// TwinCAT 3 PLC project _243401_DIOSNA_PLC
// ProgramVersion: 3.1.4026.19
// libraries:
//   Tc2_ControllerToolbox, * (Beckhoff Automation GmbH)
//   Tc2_Standard, * (Beckhoff Automation GmbH)
//   Tc2_SUPS, * (Beckhoff Automation GmbH)
//   Tc2_System, * (Beckhoff Automation GmbH)
//   Tc2_Utilities, * (Beckhoff Automation GmbH)
//   Tc3_Database, * (Beckhoff Automation GmbH)
//   Tc3_EventLogger, * (Beckhoff Automation GmbH)
//   Tc3_IPCDiag, * (Beckhoff Automation GmbH)
//   Tc3_Module, * (Beckhoff Automation GmbH)
// project tree:
//   DUTs/DataBase/ ST_BatchTrail.TcDUT, ST_ProcessData.TcDUT, ST_ShortData.TcDUT, ST_SPData.TcDUT
//   DUTs/Devices/ ST_Interface_CoilCtrl.TcDUT, ST_Interface_MotorCoilsCtrl.TcDUT, ST_Interface_MotorCtrl.TcDUT, ST_Interface_ValveCtrl.TcDUT
//   DUTs/ EN_Events.TcDUT, EN_RecipeType.TcDUT (not stored), ST_Alarm.TcDUT, ST_Batch.TcDUT, ST_Diagnostic.TcDUT, ST_HMI.TcDUT, ST_Control.TcDUT, ST_HMI_Time.TcDUT (not stored), ST_Interface_PidCtrl.TcDUT, ST_ProcessCmd2.TcDUT, ST_ProcessCmd.TcDUT, ST_PythonHandshake.TcDUT, ST_RecipeList.TcDUT (not stored), ST_RecipeSP.TcDUT, ST_Report.TcDUT, ST_RX_Python.TcDUT, ST_SeqControl.TcDUT, ST_Settings.TcDUT, ST_SP_ProcessCmd.TcDUT, ST_Time.TcDUT (not stored), ST_ToHMI.TcDUT, ST_Trend.TcDUT, ST_TX_Python.TcDUT
//   DUTs/Recipe/ ST_Cleaning_Phases.TcDUT, ST_Production_Phases.TcDUT, ST_RecipeInfo.TcDUT, ST_Recipe_Cleaning.TcDUT, ST_Recipe_Production.TcDUT
//   DUTs/ST_HMI/ ST_AlarmControl.TcDUT (not stored), ST_BatchControl.TcDUT, ST_MachineControl.TcDUT, ST_ProcessControl.TcDUT, ST_ReportControl.TcDUT
//   DUTs/ST_Mapping/ ST_EL1819.TcDUT, ST_EL2809.TcDUT, ST_EL3174.TcDUT, ST_EL4008.TcDUT, ST_EL4124.TcDUT, ST_EL9110.TcDUT
//   DUTs/ST_toHMI/ ST_EnableControl.TcDUT, ST_Header.TcDUT, ST_PID.TcDUT, ST_Prompts.TcDUT, ST_SP.TcDUT
//   FBs/Devices/ FB_AnalogInput.TcPOU, FB_AnalogOutput_v01.TcPOU, FB_AnalogOutput_v02.TcPOU, FB_CoilCtrl.TcPOU, FB_MotorCoilsCtrl.TcPOU, FB_MotorFreqCtrl.TcPOU, FB_PID.TcPOU, FB_PID_AutoTuner.TcPOU, FB_PID_Gain2Time.TcPOU, FB_PID_PWM.TcPOU, FB_TemperatureInput.TcPOU, FB_ValveCtrl32.TcPOU, FB_ValveCtrl52.TcPOU
//   FBs/ FB_AlarmDiagnostic.TcPOU, FB_AuditTrail_Write.TcPOU, FB_AVG200.TcPOU, FB_Batch.TcPOU, FB_BatchLog.TcPOU, FB_DeleteOldestFile.TcPOU, FB_FileSaveAs.TcPOU (not stored), FB_FileSaveAs_V02.TcPOU (not stored), FB_PythonScript.TcPOU, FB_Scale.TcPOU (not stored), FB_SystemDateTime.TcPOU, FB_TimeElapsed_HMI.TcPOU (not stored), FB_TONP.TcPOU (not stored)
//   Functions/ F_Interlocks.TcPOU (not stored), F_OperationalTime.TcPOU (not stored), F_Select.TcPOU, F_StepCMP.TcPOU (not stored), F_TimeBarHMI.TcPOU (not stored), F_TimerEt2String.TcPOU, F_TimerHMI.TcPOU (not stored), F_ToArrAlarms.TcPOU, F_ToArrInterlocks.TcPOU
//   GVLs/ CONST.TcGVL, GV.TcGVL, IN.TcGVL, OUT.TcGVL, Recipes.TcGVL
//   / PlcTask.TcTTO
//   POUs/0. Input/ P0_01_Mapping.TcPOU, P0_00_MAIN.TcPOU, P0_02_AnalogInput.TcPOU
//   POUs/1. Main Control/ P1_00_MAIN.TcPOU, P1_01_Recipe.TcPOU, P1_02_Batch.TcPOU, P1_03_Alarms.TcPOU, P1_04_MachineControl.TcPOU
//   POUs/2. Process/Cleaning/ _BlowingOut.TcPOU, _Control.TcPOU, _Draining.TcPOU, _MainCleaning.TcPOU, _PreCleaning.TcPOU, _PWCleaning.TcPOU, _Rinsing.TcPOU
//   POUs/2. Process/ P2_00_MAIN.TcPOU, P2_01_Production_Seq.TcPOU, P2_02_Cleaning_Seq.TcPOU, P2_03_Production_Ctrl.TcPOU, P2_04_Cleaning_Ctrl.TcPOU, P2_05_Process_Ctrl.TcPOU, P2_05_SP_Process_Ctrl.TcPOU, P2_06_Device_Ctrl.TcPOU, _Chopper.TcPOU, _FilterClean.TcPOU, _Mixer.TcPOU, _Sieve.TcPOU, _SPHeater.TcPOU, _SPMixer.TcPOU, _ToolLift.TcPOU
//   POUs/2. Process/Production/ _Discharge.TcPOU, _Feeding.TcPOU, _Granulation.TcPOU, _Mixing.TcPOU
//   POUs/3. Report/ P3_00_MAIN.TcPOU, P3_01_BatchData.TcPOU, P3_01_SP_BatchData.TcPOU, P3_03_ProcessData.TcPOU, P3_03_SP_ProcessData.TcPOU, P3_04_Alarms.TcPOU, P3_05_BatchTrail.TcPOU, P3_06_CreateReport.TcPOU, P3_06_SP_CreateReport.TcPOU, P3_07_SendReport.TcPOU, P3_08_OpenReport.TcPOU
//   POUs/5. HMI/ P5_00_MAIN.TcPOU, P5_01_EnableControls.TcPOU, P5_02_DiagramVisualisation.TcPOU, P5_03_OtherControl.TcPOU, P5_04_Trends.TcPOU
//   POUs/ MAIN.TcPOU, P02_GlobalSystemTime.TcPOU, P03_DiskSize.TcPOU, P04_Screenshot.TcPOU, SIMULATION.TcPOU
// real-time tasks:
//   TASK PlcTask: cycle T#10ms, priority 10, ADS port 350
// I/O:
//   DEVICE EtherCAT (disabled), AmsNetId 10.0.0.104.6.1
//     BUS1 (EK1100) [EK1100 EtherCAT Coupler (2A E-Bus)]
//       TI1 (EL3214) [EL3214 4K. Ana. Eingang PT100 (RTD)]
//       AI1 (EL3174) [EL3174 4Ch. Ana. Input +/-10V Diff., +/-20mA SingleEnded, 16 Bit]
//       AI2 (EL3174) [EL3174 4Ch. Ana. Input +/-10V Diff., +/-20mA SingleEnded, 16 Bit]
//       DI1 (EL1819) [EL1819 16Ch. Dig. Input 24V, 10µs]
//       DI2 (EL1819) [EL1819 16Ch. Dig. Input 24V, 10µs]
//       DI3 (EL1819) [EL1819 16Ch. Dig. Input 24V, 10µs]
//       DI4 (EL1819) [EL1819 16Ch. Dig. Input 24V, 10µs]
//       AO1 (EL4124) [EL4124 4Ch. Ana. Output 4-20mA, 16bit]
//       AO2 (EL4124) [EL4124 4Ch. Ana. Output 4-20mA, 16bit]
//       DO1 (EL2809) [EL2809 16Ch. Dig. Output 24V, 0.5A]
//       DO2 (EL2809) [EL2809 16Ch. Dig. Output 24V, 0.5A]
//       DO3 (EL2809) [EL2809 16Ch. Dig. Output 24V, 0.5A]
//       Cover (EL9011) [EL9011 End Terminal]
// variable links:
//   243401 - DIOSNA PLC/243401 - DIOSNA PLC Instance <-> EtherCAT/BUS1 (EK1100)/AI1 (EL3174)
//     PlcTask Inputs/P0_01_Mapping.AI1.Ch1_Status <-> AI Standard Channel 1/Status
//     PlcTask Inputs/P0_01_Mapping.AI1.Ch2_Status <-> AI Standard Channel 2/Status
//     PlcTask Inputs/P0_01_Mapping.AI1.Ch3_Status <-> AI Standard Channel 3/Status
//     PlcTask Inputs/P0_01_Mapping.AI1.Ch4_Status <-> AI Standard Channel 4/Status
//     PlcTask Inputs/P0_01_Mapping.AI1.Ch1_Value <-> AI Standard Channel 1/Value
//     PlcTask Inputs/P0_01_Mapping.AI1.Ch2_Value <-> AI Standard Channel 2/Value
//     PlcTask Inputs/P0_01_Mapping.AI1.Ch3_Value <-> AI Standard Channel 3/Value
//     PlcTask Inputs/P0_01_Mapping.AI1.Ch4_Value <-> AI Standard Channel 4/Value
//     PlcTask Inputs/P0_01_Mapping.AI1.State <-> InfoData/State
//   243401 - DIOSNA PLC/243401 - DIOSNA PLC Instance <-> EtherCAT/BUS1 (EK1100)/AI2 (EL3174)
//     PlcTask Inputs/P0_01_Mapping.AI2.Ch1_Status <-> AI Standard Channel 1/Status
//     PlcTask Inputs/P0_01_Mapping.AI2.Ch2_Status <-> AI Standard Channel 2/Status
//     PlcTask Inputs/P0_01_Mapping.AI2.Ch3_Status <-> AI Standard Channel 3/Status
//     PlcTask Inputs/P0_01_Mapping.AI2.Ch4_Status <-> AI Standard Channel 4/Status
//     PlcTask Inputs/P0_01_Mapping.AI2.Ch1_Value <-> AI Standard Channel 1/Value
//     PlcTask Inputs/P0_01_Mapping.AI2.Ch2_Value <-> AI Standard Channel 2/Value
//     PlcTask Inputs/P0_01_Mapping.AI2.Ch3_Value <-> AI Standard Channel 3/Value
//     PlcTask Inputs/P0_01_Mapping.AI2.Ch4_Value <-> AI Standard Channel 4/Value
//     PlcTask Inputs/P0_01_Mapping.AI2.State <-> InfoData/State
//   243401 - DIOSNA PLC/243401 - DIOSNA PLC Instance <-> EtherCAT/BUS1 (EK1100)/AO1 (EL4124)
//     PlcTask Inputs/P0_01_Mapping.AO1.State <-> InfoData/State
//     PlcTask Outputs/P0_01_Mapping.AO1.Ch1_Value <-> AO Output Channel 1/Analog output
//     PlcTask Outputs/P0_01_Mapping.AO1.Ch2_Value <-> AO Output Channel 2/Analog output
//     PlcTask Outputs/P0_01_Mapping.AO1.Ch3_Value <-> AO Output Channel 3/Analog output
//     PlcTask Outputs/P0_01_Mapping.AO1.Ch4_Value <-> AO Output Channel 4/Analog output
//   243401 - DIOSNA PLC/243401 - DIOSNA PLC Instance <-> EtherCAT/BUS1 (EK1100)/AO2 (EL4124)
//     PlcTask Inputs/P0_01_Mapping.AO2.State <-> InfoData/State
//     PlcTask Outputs/P0_01_Mapping.AO2.Ch1_Value <-> AO Output Channel 1/Analog output
//     PlcTask Outputs/P0_01_Mapping.AO2.Ch2_Value <-> AO Output Channel 2/Analog output
//     PlcTask Outputs/P0_01_Mapping.AO2.Ch3_Value <-> AO Output Channel 3/Analog output
//     PlcTask Outputs/P0_01_Mapping.AO2.Ch4_Value <-> AO Output Channel 4/Analog output
//   243401 - DIOSNA PLC/243401 - DIOSNA PLC Instance <-> EtherCAT/BUS1 (EK1100)/DI1 (EL1819)
//     PlcTask Inputs/P0_01_Mapping.DI1.Ch10_Value <-> Channel 10/Input
//     PlcTask Inputs/P0_01_Mapping.DI1.Ch11_Value <-> Channel 11/Input
//     PlcTask Inputs/P0_01_Mapping.DI1.Ch12_Value <-> Channel 12/Input
//     PlcTask Inputs/P0_01_Mapping.DI1.Ch13_Value <-> Channel 13/Input
//     PlcTask Inputs/P0_01_Mapping.DI1.Ch14_Value <-> Channel 14/Input
//     PlcTask Inputs/P0_01_Mapping.DI1.Ch15_Value <-> Channel 15/Input
//     PlcTask Inputs/P0_01_Mapping.DI1.Ch16_Value <-> Channel 16/Input
//     PlcTask Inputs/P0_01_Mapping.DI1.Ch1_Value <-> Channel 1/Input
//     PlcTask Inputs/P0_01_Mapping.DI1.Ch2_Value <-> Channel 2/Input
//     PlcTask Inputs/P0_01_Mapping.DI1.Ch3_Value <-> Channel 3/Input
//     PlcTask Inputs/P0_01_Mapping.DI1.Ch4_Value <-> Channel 4/Input
//     PlcTask Inputs/P0_01_Mapping.DI1.Ch5_Value <-> Channel 5/Input
//     PlcTask Inputs/P0_01_Mapping.DI1.Ch6_Value <-> Channel 6/Input
//     PlcTask Inputs/P0_01_Mapping.DI1.Ch7_Value <-> Channel 7/Input
//     PlcTask Inputs/P0_01_Mapping.DI1.Ch8_Value <-> Channel 8/Input
//     PlcTask Inputs/P0_01_Mapping.DI1.Ch9_Value <-> Channel 9/Input
//     PlcTask Inputs/P0_01_Mapping.DI1.State <-> InfoData/State
//   243401 - DIOSNA PLC/243401 - DIOSNA PLC Instance <-> EtherCAT/BUS1 (EK1100)/DI2 (EL1819)
//     PlcTask Inputs/P0_01_Mapping.DI2.Ch10_Value <-> Channel 10/Input
//     PlcTask Inputs/P0_01_Mapping.DI2.Ch11_Value <-> Channel 11/Input
//     PlcTask Inputs/P0_01_Mapping.DI2.Ch12_Value <-> Channel 12/Input
//     PlcTask Inputs/P0_01_Mapping.DI2.Ch13_Value <-> Channel 13/Input
//     PlcTask Inputs/P0_01_Mapping.DI2.Ch14_Value <-> Channel 14/Input
//     PlcTask Inputs/P0_01_Mapping.DI2.Ch15_Value <-> Channel 15/Input
//     PlcTask Inputs/P0_01_Mapping.DI2.Ch16_Value <-> Channel 16/Input
//     PlcTask Inputs/P0_01_Mapping.DI2.Ch1_Value <-> Channel 1/Input
//     PlcTask Inputs/P0_01_Mapping.DI2.Ch2_Value <-> Channel 2/Input
//     PlcTask Inputs/P0_01_Mapping.DI2.Ch3_Value <-> Channel 3/Input
//     PlcTask Inputs/P0_01_Mapping.DI2.Ch4_Value <-> Channel 4/Input
//     PlcTask Inputs/P0_01_Mapping.DI2.Ch5_Value <-> Channel 5/Input
//     PlcTask Inputs/P0_01_Mapping.DI2.Ch6_Value <-> Channel 6/Input
//     PlcTask Inputs/P0_01_Mapping.DI2.Ch7_Value <-> Channel 7/Input
//     PlcTask Inputs/P0_01_Mapping.DI2.Ch8_Value <-> Channel 8/Input
//     PlcTask Inputs/P0_01_Mapping.DI2.Ch9_Value <-> Channel 9/Input
//     PlcTask Inputs/P0_01_Mapping.DI2.State <-> InfoData/State
//   243401 - DIOSNA PLC/243401 - DIOSNA PLC Instance <-> EtherCAT/BUS1 (EK1100)/DI3 (EL1819)
//     PlcTask Inputs/P0_01_Mapping.DI3.Ch10_Value <-> Channel 10/Input
//     PlcTask Inputs/P0_01_Mapping.DI3.Ch11_Value <-> Channel 11/Input
//     PlcTask Inputs/P0_01_Mapping.DI3.Ch12_Value <-> Channel 12/Input
//     PlcTask Inputs/P0_01_Mapping.DI3.Ch13_Value <-> Channel 13/Input
//     PlcTask Inputs/P0_01_Mapping.DI3.Ch14_Value <-> Channel 14/Input
//     PlcTask Inputs/P0_01_Mapping.DI3.Ch15_Value <-> Channel 15/Input
//     PlcTask Inputs/P0_01_Mapping.DI3.Ch16_Value <-> Channel 16/Input
//     PlcTask Inputs/P0_01_Mapping.DI3.Ch1_Value <-> Channel 1/Input
//     PlcTask Inputs/P0_01_Mapping.DI3.Ch2_Value <-> Channel 2/Input
//     PlcTask Inputs/P0_01_Mapping.DI3.Ch3_Value <-> Channel 3/Input
//     PlcTask Inputs/P0_01_Mapping.DI3.Ch4_Value <-> Channel 4/Input
//     PlcTask Inputs/P0_01_Mapping.DI3.Ch5_Value <-> Channel 5/Input
//     PlcTask Inputs/P0_01_Mapping.DI3.Ch6_Value <-> Channel 6/Input
//     PlcTask Inputs/P0_01_Mapping.DI3.Ch7_Value <-> Channel 7/Input
//     PlcTask Inputs/P0_01_Mapping.DI3.Ch8_Value <-> Channel 8/Input
//     PlcTask Inputs/P0_01_Mapping.DI3.Ch9_Value <-> Channel 9/Input
//     PlcTask Inputs/P0_01_Mapping.DI3.State <-> InfoData/State
//   243401 - DIOSNA PLC/243401 - DIOSNA PLC Instance <-> EtherCAT/BUS1 (EK1100)/DI4 (EL1819)
//     PlcTask Inputs/P0_01_Mapping.DI4.Ch10_Value <-> Channel 10/Input
//     PlcTask Inputs/P0_01_Mapping.DI4.Ch11_Value <-> Channel 11/Input
//     PlcTask Inputs/P0_01_Mapping.DI4.Ch12_Value <-> Channel 12/Input
//     PlcTask Inputs/P0_01_Mapping.DI4.Ch13_Value <-> Channel 13/Input
//     PlcTask Inputs/P0_01_Mapping.DI4.Ch14_Value <-> Channel 14/Input
//     PlcTask Inputs/P0_01_Mapping.DI4.Ch15_Value <-> Channel 15/Input
//     PlcTask Inputs/P0_01_Mapping.DI4.Ch16_Value <-> Channel 16/Input
//     PlcTask Inputs/P0_01_Mapping.DI4.Ch1_Value <-> Channel 1/Input
//     PlcTask Inputs/P0_01_Mapping.DI4.Ch2_Value <-> Channel 2/Input
//     PlcTask Inputs/P0_01_Mapping.DI4.Ch3_Value <-> Channel 3/Input
//     PlcTask Inputs/P0_01_Mapping.DI4.Ch4_Value <-> Channel 4/Input
//     PlcTask Inputs/P0_01_Mapping.DI4.Ch5_Value <-> Channel 5/Input
//     PlcTask Inputs/P0_01_Mapping.DI4.Ch6_Value <-> Channel 6/Input
//     PlcTask Inputs/P0_01_Mapping.DI4.Ch7_Value <-> Channel 7/Input
//     PlcTask Inputs/P0_01_Mapping.DI4.Ch8_Value <-> Channel 8/Input
//     PlcTask Inputs/P0_01_Mapping.DI4.Ch9_Value <-> Channel 9/Input
//     PlcTask Inputs/P0_01_Mapping.DI4.State <-> InfoData/State
//   243401 - DIOSNA PLC/243401 - DIOSNA PLC Instance <-> EtherCAT/BUS1 (EK1100)/DO1 (EL2809)
//     PlcTask Inputs/P0_01_Mapping.DO1.State <-> InfoData/State
//     PlcTask Outputs/P0_01_Mapping.DO1.Ch10_Value <-> Channel 10/Output
//     PlcTask Outputs/P0_01_Mapping.DO1.Ch11_Value <-> Channel 11/Output
//     PlcTask Outputs/P0_01_Mapping.DO1.Ch12_Value <-> Channel 12/Output
//     PlcTask Outputs/P0_01_Mapping.DO1.Ch13_Value <-> Channel 13/Output
//     PlcTask Outputs/P0_01_Mapping.DO1.Ch14_Value <-> Channel 14/Output
//     PlcTask Outputs/P0_01_Mapping.DO1.Ch15_Value <-> Channel 15/Output
//     PlcTask Outputs/P0_01_Mapping.DO1.Ch16_Value <-> Channel 16/Output
//     PlcTask Outputs/P0_01_Mapping.DO1.Ch1_Value <-> Channel 1/Output
//     PlcTask Outputs/P0_01_Mapping.DO1.Ch2_Value <-> Channel 2/Output
//     PlcTask Outputs/P0_01_Mapping.DO1.Ch3_Value <-> Channel 3/Output
//     PlcTask Outputs/P0_01_Mapping.DO1.Ch4_Value <-> Channel 4/Output
//     PlcTask Outputs/P0_01_Mapping.DO1.Ch5_Value <-> Channel 5/Output
//     PlcTask Outputs/P0_01_Mapping.DO1.Ch6_Value <-> Channel 6/Output
//     PlcTask Outputs/P0_01_Mapping.DO1.Ch7_Value <-> Channel 7/Output
//     PlcTask Outputs/P0_01_Mapping.DO1.Ch8_Value <-> Channel 8/Output
//     PlcTask Outputs/P0_01_Mapping.DO1.Ch9_Value <-> Channel 9/Output
//   243401 - DIOSNA PLC/243401 - DIOSNA PLC Instance <-> EtherCAT/BUS1 (EK1100)/DO2 (EL2809)
//     PlcTask Inputs/P0_01_Mapping.DO2.State <-> InfoData/State
//     PlcTask Outputs/P0_01_Mapping.DO2.Ch10_Value <-> Channel 10/Output
//     PlcTask Outputs/P0_01_Mapping.DO2.Ch11_Value <-> Channel 11/Output
//     PlcTask Outputs/P0_01_Mapping.DO2.Ch12_Value <-> Channel 12/Output
//     PlcTask Outputs/P0_01_Mapping.DO2.Ch13_Value <-> Channel 13/Output
//     PlcTask Outputs/P0_01_Mapping.DO2.Ch14_Value <-> Channel 14/Output
//     PlcTask Outputs/P0_01_Mapping.DO2.Ch15_Value <-> Channel 15/Output
//     PlcTask Outputs/P0_01_Mapping.DO2.Ch16_Value <-> Channel 16/Output
//     PlcTask Outputs/P0_01_Mapping.DO2.Ch1_Value <-> Channel 1/Output
//     PlcTask Outputs/P0_01_Mapping.DO2.Ch2_Value <-> Channel 2/Output
//     PlcTask Outputs/P0_01_Mapping.DO2.Ch3_Value <-> Channel 3/Output
//     PlcTask Outputs/P0_01_Mapping.DO2.Ch4_Value <-> Channel 4/Output
//     PlcTask Outputs/P0_01_Mapping.DO2.Ch5_Value <-> Channel 5/Output
//     PlcTask Outputs/P0_01_Mapping.DO2.Ch6_Value <-> Channel 6/Output
//     PlcTask Outputs/P0_01_Mapping.DO2.Ch7_Value <-> Channel 7/Output
//     PlcTask Outputs/P0_01_Mapping.DO2.Ch8_Value <-> Channel 8/Output
//     PlcTask Outputs/P0_01_Mapping.DO2.Ch9_Value <-> Channel 9/Output
//   243401 - DIOSNA PLC/243401 - DIOSNA PLC Instance <-> EtherCAT/BUS1 (EK1100)/DO3 (EL2809)
//     PlcTask Inputs/P0_01_Mapping.DO3.State <-> InfoData/State
//     PlcTask Outputs/P0_01_Mapping.DO3.Ch10_Value <-> Channel 10/Output
//     PlcTask Outputs/P0_01_Mapping.DO3.Ch11_Value <-> Channel 11/Output
//     PlcTask Outputs/P0_01_Mapping.DO3.Ch12_Value <-> Channel 12/Output
//     PlcTask Outputs/P0_01_Mapping.DO3.Ch13_Value <-> Channel 13/Output
//     PlcTask Outputs/P0_01_Mapping.DO3.Ch14_Value <-> Channel 14/Output
//     PlcTask Outputs/P0_01_Mapping.DO3.Ch15_Value <-> Channel 15/Output
//     PlcTask Outputs/P0_01_Mapping.DO3.Ch16_Value <-> Channel 16/Output
//     PlcTask Outputs/P0_01_Mapping.DO3.Ch1_Value <-> Channel 1/Output
//     PlcTask Outputs/P0_01_Mapping.DO3.Ch2_Value <-> Channel 2/Output
//     PlcTask Outputs/P0_01_Mapping.DO3.Ch3_Value <-> Channel 3/Output
//     PlcTask Outputs/P0_01_Mapping.DO3.Ch4_Value <-> Channel 4/Output
//     PlcTask Outputs/P0_01_Mapping.DO3.Ch5_Value <-> Channel 5/Output
//     PlcTask Outputs/P0_01_Mapping.DO3.Ch6_Value <-> Channel 6/Output
//     PlcTask Outputs/P0_01_Mapping.DO3.Ch7_Value <-> Channel 7/Output
//     PlcTask Outputs/P0_01_Mapping.DO3.Ch8_Value <-> Channel 8/Output
//     PlcTask Outputs/P0_01_Mapping.DO3.Ch9_Value <-> Channel 9/Output

CONFIGURATION _243401_DIOSNA_PLC
    RESOURCE PLC ON TwinCAT3
        TASK PlcTask(INTERVAL := T#10ms, PRIORITY := 10);
        PROGRAM MAIN WITH PlcTask : MAIN;
    END_RESOURCE
END_CONFIGURATION

// ---- DUTs/DataBase/ST_BatchTrail.TcDUT
TYPE ST_BatchTrail :
STRUCT
	Batch				:STRING(100);
	Event				:STRING(100);
	Description			:STRING(100);
	User				:STRING(100);
	Oldvalue			:STRING(100);
	Newvalue			:STRING(100);
END_STRUCT
END_TYPE

// ---- DUTs/DataBase/ST_ProcessData.TcDUT
TYPE ST_ProcessData :
STRUCT
	batch		: STRING(100);
	number		: STRING(100);
	name		: STRING(100);
	value1		: REAL; 
	value2		: REAL;
	value3		: REAL;
	value4		: REAL;
	value5 		: REAL;
	value6		: REAL; 
END_STRUCT
END_TYPE

// ---- DUTs/DataBase/ST_ShortData.TcDUT
TYPE ST_ShortData :
STRUCT
	Batch		: STRING(100);
	Number		: STRING(100);
	Name		: STRING(100);
	Event		: STRING(100);
	DateTime	: DT;
END_STRUCT
END_TYPE

// ---- DUTs/DataBase/ST_SPData.TcDUT
TYPE ST_SPData :
STRUCT
	Value1		: STRING(100);
	Value2		: STRING(100);
	Value3		: STRING(100);
	DateTime	: DT;
END_STRUCT
END_TYPE

// ---- DUTs/Devices/ST_Interface_CoilCtrl.TcDUT
TYPE ST_Interface_CoilCtrl :
STRUCT
	//IN
	arrInterlocks		:ARRAY[1..8] OF BOOL;
	arrAlarms			:ARRAY[1..8] OF BOOL;
	bCmd				:BOOL;
	bServiceMode		:BOOL;
	iMaintLimit			:UDINT;
	iPresetValue		:UDINT;
	bWritePreset		:BOOL;
	//OUT
	bInterlocksOK		:BOOL;
	bCmdOut				:BOOL;
	bFault				:BOOL;
	iTotalCycles		:UDINT;
	iMaintCycles		:UDINT;
	bMaintCall			:BOOL;
END_STRUCT
END_TYPE

// ---- DUTs/Devices/ST_Interface_MotorCoilsCtrl.TcDUT
TYPE ST_Interface_MotorCoilsCtrl :
STRUCT
	//IN
	arrInterlocks		:ARRAY[1..8] OF BOOL;
	arrAlarms			:ARRAY[1..8] OF BOOL;
	bCmdSlow			:BOOL;
	bCmdFast			:BOOL;
	bCmdStop			:BOOL;
	rSlowSpeed			:REAL;
	rFastSpeed			:REAL;
	rFeedback1			:REAL;
	rFeedback2			:REAL;
	bEnableMonitor		:BOOL;
	iMonitorTime		:INT;
	iMonitorTolerance	:INT;
	bServiceMode		:BOOL;
	iMaintLimit			:REAL;
	iPresetValue		:REAL;
	bWritePreset		:BOOL;
	//OUT
	bInterlocksOK		:BOOL;
	bCmdOutSlow			:BOOL;
	bCmdOutFast			:BOOL;
	bFault				:BOOL;
	iTotalHours			:REAL;
	iMaintHours			:REAL;
	bMaintCall			:BOOL;	
	iState				:INT;
END_STRUCT
END_TYPE

// ---- DUTs/Devices/ST_Interface_MotorCtrl.TcDUT
TYPE ST_Interface_MotorCtrl :
STRUCT
	//IN
	arrInterlocks		:ARRAY[1..8] OF BOOL;
	arrAlarms			:ARRAY[1..8] OF BOOL;
	bCmdBwd				:BOOL;
	bCmdFwd				:BOOL;
	bCmdStop			:BOOL;
	iSetpoint			:INT;
	rFeedback1			:REAL;
	rFeedback2			:REAL;
	bEnableMonitor		:BOOL;
	iMonitorTime		:INT;
	iMonitorTolerance	:INT;
	bServiceMode		:BOOL;
	iMaintLimit			:REAL;
	iPresetValue		:REAL;
	bWritePreset		:BOOL;
	//OUT
	bInterlocksOK		:BOOL;
	bCmdOutBwd			:BOOL;
	bCmdOutFwd			:BOOL;
	bFault				:BOOL;
	iTotalHours			:REAL;
	iMaintHours			:REAL;
	bMaintCall			:BOOL;	
	iState				:INT;
END_STRUCT
END_TYPE

// ---- DUTs/Devices/ST_Interface_ValveCtrl.TcDUT
TYPE ST_Interface_ValveCtrl :
STRUCT
	//IN
	arrInterlocks		:ARRAY[1..8] OF BOOL;
	arrAlarms			:ARRAY[1..8] OF BOOL;
	bCmdHP				:BOOL;
	bCmdWP				:BOOL;
	bEnableHP			:BOOL;
	bEnableWP			:BOOL;
	iTravelTimeout		:INT;
	bServiceMode		:BOOL;
	iMaintLimit			:UDINT;
	iPresetValue		:UDINT;
	bWritePreset		:BOOL;
	//OUT
	bInterlocksOK		:BOOL;
	bCmdOutHP			:BOOL;
	bCmdOutWP			:BOOL;
	bFault				:BOOL;
	iTotalCycles		:UDINT;
	iMaintCycles		:UDINT;
	bMaintCall			:BOOL;
	iState				:INT;
END_STRUCT
END_TYPE

// ---- DUTs/EN_Events.TcDUT
{attribute 'to_string'}
TYPE EN_Events :
(
	NOT_DEFINED		:= 0,
	RECIPE		    := 1,
	BATCH			:= 2,
	GENERAL			:= 3,
	SETTINGS		:= 4,
	SP				:= 5		
);
END_TYPE

// ---- DUTs/Recipe/ST_Cleaning_Phases.TcDUT
TYPE ST_Cleaning_Phases :
STRUCT
	bEnable								:BOOL;
	iType								:INT;  //0-Pre-Cleaning, 1-Main Clean, 2-Rinse, 3-PW Clean, 4 - Draining, 5 Blowing out, 6 - Control
	sDescription						:STRING;
	iChopper							:INT;  //0-OFF,1-ON
	rMixerSpeed1						:REAL; //Mixer speed during filling
	rMixerSpeed2						:REAL; //Mixer speed during mixing
	rMixerSpeed3						:REAL; //Mixer speed during emptying
	rSieveSpeed							:REAL; //Sieve speed
	iMedium								:INT;  //0-Cold water,1-Warm water
	iDetergent							:INT;  //0-OFF,1-ON
	bMixerWater							:BOOL; //Fill water from mixer
	bChopperWater						:BOOL; //Fill water fromo choper
	bSPWater							:BOOL; //Fill water in SP
	iTime1								:ST_HMI_Time;			
	iTime2								:ST_HMI_Time;
	iTime3								:ST_HMI_Time;
END_STRUCT
END_TYPE

// ---- DUTs/Recipe/ST_Production_Phases.TcDUT
TYPE ST_Production_Phases :
STRUCT
	bEnable					:BOOL;
	iType					:INT;  				//0-Feeding,1-Mixing,2-Granulation,3-Discharge
	sDescription			:STRING;		
	iEndPoint				:INT;    			//0-Manual,1-Auto,2-Mixer current
	iPhaseTime				:ST_HMI_Time;		//min:sec
	iFilterClean			:DINT;				//sec
	iFilterPause			:DINT;				//sec
	iMixer					:INT;				//0-off,1-on
	rMixerSpeed				:REAL;				//rpm
	rMixerCurrent			:REAL;				//A
	iChopper				:INT;				//0-OFF,1-Slow,2-Fast
	rSieveSpeed				:REAL;				//rpm
	bPause					:BOOL;				//0-continue,1-pause
	rSP_MixingSpeed			:REAL;
	rSP_Temperature			:REAL;
	rSP_Pressure			:REAL;
END_STRUCT
END_TYPE

// ---- DUTs/Recipe/ST_RecipeInfo.TcDUT
TYPE ST_RecipeInfo :
STRUCT
	sUserCreated		:STRING;
	sUserEdited			:STRING;
	sUserVerified		:STRING;
	sTimeCreated		:STRING;
	sTimeEdited			:STRING;
	sTimeVerified		:STRING;
	bVerification		:BOOL;
	iVersion			:INT;
END_STRUCT
END_TYPE

// ---- DUTs/Recipe/ST_Recipe_Cleaning.TcDUT
TYPE ST_Recipe_Cleaning :
STRUCT
	sName					:STRING[80];
	stInfo					:ST_RecipeInfo;
	stPhase					:ARRAY[0..20] OF ST_Cleaning_Phases;
	iType					:INT; 
	iActivePhase			:INT;
END_STRUCT
END_TYPE

// ---- DUTs/Recipe/ST_Recipe_Production.TcDUT
TYPE ST_Recipe_Production :
STRUCT
	sName					:STRING[80];
	stInfo					:ST_RecipeInfo;
	stPhase					:ARRAY[0..20] OF ST_Production_Phases;
	iType					:INT; 
	iActivePhase			:INT;
END_STRUCT
END_TYPE

// ---- DUTs/ST_Alarm.TcDUT
TYPE ST_Alarm :
STRUCT
	Alarm			:ARRAY[0..99] OF fb_TcAlarm;
	Active			:ARRAY[0..99] OF BOOL;
	Raise			:ARRAY[0..99] OF BOOL;
	
END_STRUCT
END_TYPE

// ---- DUTs/ST_Batch.TcDUT
TYPE ST_Batch :
STRUCT
	sBatchNumber		:STRING;
	sBatchName			:STRING;
	sRecipeName			:STRING;
	sRecipeType			:STRING;
	sProductName		:STRING;
	sComment			:STRING;
	sUser				:STRING;
	sStarted			:STRING;
	sFinished			:STRING;
END_STRUCT
END_TYPE

// ---- DUTs/ST_Diagnostic.TcDUT
TYPE ST_Diagnostic :
STRUCT
	Temperature			:UDINT;
	BootCount			:UDINT;
	OperationTime		:UDINT;
	OperationDuration	:ARRAY[0..2] OF INT;
END_STRUCT
END_TYPE

// ---- DUTs/ST_HMI.TcDUT
TYPE ST_HMI :
STRUCT
	
	stMachine_Ctrl						:ST_MachineControl;
	stSP_Machine_Ctrl					:ST_MachineControl;
	stBatch_Ctrl						:ST_BatchControl;

	stReport_Ctrl						:ST_ReportControl;
	stProcess_Ctrl						:ST_ProcessControl;
	stAlarm_Ctrl						:ST_AlarmControl;
	
	iSelectedPhase						:INT;
	bCloseHMI							:BOOL;
	bScreenshot							:BOOL;
	bScanBatchParams					:BOOL;
	bReadCapacity						:BOOL;
		
END_STRUCT
END_TYPE

// ---- DUTs/ST_HMI/ST_BatchControl.TcDUT
TYPE ST_BatchControl :
STRUCT
	bCreate			:BOOL;
	bCancel			:BOOL;
	bOpen			:BOOL;
	bClose			:BOOL;
	bLoad			:BOOL;
	bLoadSP			:BOOL;
	
	sName			:STRING;
	sNameSP			:STRING;
	iNumber			:UDINT;
	iSubNumber		:INT;
	sProduct		:STRING;
	sComment		:STRING;
	sRecipe			:STRING;
	sRecipeSP		:STRING;
	
	iRecipeType		:INT;
	iSelectedPhase	:INT;
END_STRUCT
END_TYPE

// ---- DUTs/ST_HMI/ST_MachineControl.TcDUT
TYPE ST_MachineControl :
STRUCT
	bAuto					:BOOL;
	bService				:BOOL;
	bStart					:BOOL;
	bStop					:BOOL;
	bPause					:BOOL;
	bNext					:BOOL;
	bPrevious				:BOOL;
	bJump					:BOOL;
	bLogIn					:BOOL;
END_STRUCT
END_TYPE

// ---- DUTs/ST_HMI/ST_ProcessControl.TcDUT
TYPE ST_ProcessControl :
STRUCT

	bLid_Open						:BOOL;
	bLid_Close						:BOOL;
	bOutlet_Open					:BOOL;
	bOutlet_Close					:BOOL;
	bSieve_SealOn					:BOOL;
	bSieve_SealOff					:BOOL;
	bTool_Raise						:BOOL;
	bTool_Lower						:BOOL;
	bMixer_FindPos					:BOOL;
	
	bPump_Start						:BOOL;
	bPump_Stop						:BOOL;
	bMixer_Start					:BOOL;
	bMixer_Stop						:BOOL;
	bSieve_Start					:BOOL;
	bSieve_Stop						:BOOL;
	
	bSP_Mixer_Toggle				:BOOL;
	bSP_Heater_Toggle				:BOOL;
	
	
	bConfirm_Prompt					:BOOL;
	bConfirm_IsClean				:BOOL;
	bConfirm_NotClean				:BOOL;
END_STRUCT
END_TYPE

// ---- DUTs/ST_HMI/ST_ReportControl.TcDUT
TYPE ST_ReportControl :
STRUCT
	iIndex					:INT;
	iReportOpen				:INT;
	bProcessReport			:BOOL;
END_STRUCT
END_TYPE

// ---- DUTs/ST_Control.TcDUT
TYPE ST_Control :
STRUCT
	bAbort					:BOOL;
	bRunning				:BOOL;
	bNext					:BOOL;
	bPrevious				:BOOL;
	bAuto					:BOOL;
	bRecovery				:BOOL;
	bServiceMode			:BOOL;
	bFinish					:BOOL;
	bPaused					:BOOL;
	bStopped				:BOOL;
	bPhaseFinished			:BOOL;
	bPhasePaused			:BOOL;
	bIntelrockOK			:BOOL;
	bProcesslockOK			:BOOL;
	bConfirmation			:BOOL;
	bOperation				:BOOL;
	bJump					:BOOL;
	bStarting				:BOOL;
	bStopping				:BOOL;
	iJumpStep				:INT;
END_STRUCT
END_TYPE

// ---- DUTs/ST_Interface_PidCtrl.TcDUT
TYPE ST_Interface_PidCtrl :
STRUCT
	//Input
	i_bEnablePID		:BOOL;
	i_rSetpoint			:REAL;
	i_rActual			:REAL;
	i_rKp				:REAL;
	i_rKi				:REAL;
	i_rKd				:REAL;
	i_rTdamp			:REAL;
	i_rOutMin			:REAL;
	i_rOutMax			:REAL;
	i_rManualOutput		:REAL;
	i_bEnablePWM		:BOOL;
	i_iFreqPWM			:INT;
	i_bAutotuneStart	:BOOL;
	i_rAutotuneSetpoint	:REAL;
	i_bAutotuneAccept	:BOOL;
	i_bEnableAlarms		:BOOL;
	i_iHighAlarm		:INT;
	i_iHighWarning		:INT;
	i_iLowWarning		:INT;
	i_iLowAlarm			:INT;
	i_iWarningDelay		:INT;
	i_iAlarmDelay		:INT;
	//Output
	q_rOutputPID		:REAL;
	q_bOutputPWM		:BOOL;
	q_Difference		:REAL;
	q_AutotuneActive	:BOOL;
	q_AutotuneDone		:BOOL;
	i_sAutotuneTime		:STRING;
	q_rAutotuneKp		:REAL;
	q_rAutotuneKi		:REAL;
	q_rAutotuneKd		:REAL;
	q_bError			:BOOL;
	q_bErrorID			:INT;
	q_bAlarmHigh		:BOOL;
	q_bWarningHigh		:BOOL;
	q_bWarningLow		:BOOL;
	q_bAlarmLow			:BOOL;
END_STRUCT
END_TYPE

// ---- DUTs/ST_ProcessCmd2.TcDUT
TYPE ST_ProcessCmd2 :
STRUCT
	bLid_Open			:BOOL;
	bLid_Close			:BOOL;
	bOutlet_Open		:BOOL;
	bOutlet_Close		:BOOL;
	bSieveSeal_Off		:BOOL;
	bSieveSeal_On		:BOOL;
	bTool_Raise			:BOOL;
	bTool_Lower			:BOOL;
	bPurge_Max			:BOOL;
	bPurge_Min			:BOOL;
END_STRUCT
END_TYPE

// ---- DUTs/ST_Mapping/ST_EL1819.TcDUT
TYPE ST_EL1819 :
STRUCT
	Ch1_Value						AT %I*	:BOOL;
	Ch2_Value						AT %I*	:BOOL;
	Ch3_Value						AT %I*	:BOOL;
	Ch4_Value						AT %I*	:BOOL;
	Ch5_Value						AT %I*	:BOOL;
	Ch6_Value						AT %I*	:BOOL;
	Ch7_Value						AT %I*	:BOOL;
	Ch8_Value						AT %I*	:BOOL;
	Ch9_Value						AT %I*	:BOOL;
	Ch10_Value						AT %I*	:BOOL;
	Ch11_Value						AT %I*	:BOOL;
	Ch12_Value						AT %I*	:BOOL;
	Ch13_Value						AT %I*	:BOOL;
	Ch14_Value						AT %I*	:BOOL;
	Ch15_Value						AT %I*	:BOOL;
	Ch16_Value						AT %I*	:BOOL;
	State							AT %I*	:UINT;
END_STRUCT
END_TYPE

// ---- DUTs/ST_Mapping/ST_EL2809.TcDUT
TYPE ST_EL2809 :
STRUCT
	Ch1_Value						AT %Q*	:BOOL;
	Ch2_Value						AT %Q*	:BOOL;
	Ch3_Value						AT %Q*	:BOOL;
	Ch4_Value						AT %Q*	:BOOL;
	Ch5_Value						AT %Q*	:BOOL;
	Ch6_Value						AT %Q*	:BOOL;
	Ch7_Value						AT %Q*	:BOOL;
	Ch8_Value						AT %Q*	:BOOL;
	Ch9_Value						AT %Q*	:BOOL;
	Ch10_Value						AT %Q*	:BOOL;
	Ch11_Value						AT %Q*	:BOOL;
	Ch12_Value						AT %Q*	:BOOL;
	Ch13_Value						AT %Q*	:BOOL;
	Ch14_Value						AT %Q*	:BOOL;
	Ch15_Value						AT %Q*	:BOOL;
	Ch16_Value						AT %Q*	:BOOL;
	State							AT %I*	:UINT;
END_STRUCT
END_TYPE

// ---- DUTs/ST_Mapping/ST_EL3174.TcDUT
TYPE ST_EL3174 :
STRUCT
	Ch1_Status						AT %I*	:Status_7EBB4A47_Plc;
	Ch1_Value						AT %I*	:INT;
	Ch2_Status						AT %I*	:Status_7EBB4A47_Plc;
	Ch2_Value						AT %I*	:INT;
	Ch3_Status						AT %I*	:Status_7EBB4A47_Plc;
	Ch3_Value						AT %I*	:INT;
	Ch4_Status						AT %I*	:Status_7EBB4A47_Plc;
	Ch4_Value						AT %I*	:INT;
	State							AT %I*	:UINT;
END_STRUCT
END_TYPE

// ---- DUTs/ST_Mapping/ST_EL4008.TcDUT
TYPE ST_EL4008 :
STRUCT
	Ch1_Value						AT %Q*	:INT;
	Ch2_Value						AT %Q*	:INT;
	Ch3_Value						AT %Q*	:INT;
	Ch4_Value						AT %Q*	:INT;
	Ch5_Value						AT %Q*	:INT;
	Ch6_Value						AT %Q*	:INT;
	Ch7_Value						AT %Q*	:INT;
	Ch8_Value						AT %Q*	:INT;
	State							AT %I*	:UINT;
END_STRUCT
END_TYPE

// ---- DUTs/ST_Mapping/ST_EL4124.TcDUT
TYPE ST_EL4124 :
STRUCT
	Ch1_Value						AT %Q*	:INT;
	Ch2_Value						AT %Q*	:INT;
	Ch3_Value						AT %Q*	:INT;
	Ch4_Value						AT %Q*	:INT;
	State							AT %I*	:UINT;
END_STRUCT
END_TYPE

// ---- DUTs/ST_Mapping/ST_EL9110.TcDUT
TYPE ST_EL9110 :
STRUCT
	PowerOK							AT %I*	:BOOL;
	State							AT %I*	:UINT;
END_STRUCT
END_TYPE

// ---- DUTs/ST_ProcessCmd.TcDUT
TYPE ST_ProcessCmd :
STRUCT
	
	bAspiration				:BOOL;	

	bOutletOpen				:BOOL;
	bOutletClose			:BOOL;
	
	rMixerSpeed				:REAL;
	bMixerStart				:BOOL;
	bMixerAir				:BOOL;
	bChopperAir				:BOOL;
	iChopper				:INT;
	rSieveSpeed				:REAL;
	bSieveStart				:BOOL;
	
	bVacuumValve			:BOOL;
	bVacuumPump				:BOOL;
	bFilterClean			:BOOL;
		
	bColdWater				:BOOL;
	bWarmWater				:BOOL;
	bPurifiedWater			:BOOL;
	bCompressedAir			:BOOL;
	
	bMixerWater				:BOOL;
	bChopperWater			:BOOL;
	bSPWater				:BOOL;
	
	bMainDrain				:BOOL;
	bSPDrain				:BOOL;
	
	bMixer					:BOOL;
	bSieve					:BOOL;
	bChopperSlow			:BOOL;
	bChopperFast			:BOOL;
	
	rSP_Pressure			:REAL;
END_STRUCT
END_TYPE

// ---- DUTs/ST_PythonHandshake.TcDUT
TYPE ST_PythonHandshake :
STRUCT
	bBusy					:BOOL;
	bDone					:BOOL;
	bError					:BOOL;
	sError					:STRING(255);
END_STRUCT
END_TYPE

// ---- DUTs/ST_RecipeSP.TcDUT
TYPE ST_RecipeSP :
STRUCT
	rMixingSpeed				:REAL;
	rTemperature				:REAL;
	stProcessTime				:ST_HMI_Time;
END_STRUCT
END_TYPE

// ---- DUTs/ST_Report.TcDUT
TYPE ST_Report :
STRUCT
	bStartCreate_Sequence				:BOOL;
	bStartSend_Sequence					:BOOL;
	bSend_Report						:BOOL;
	bExport_Alarms						:BOOL;
	bSaveAs_Alarms						:BOOL;
	bCreate_Report						:BOOL;
	bDelete_Data						:BOOL;
	bDelete_SPData						:BOOL;
	bDelete_OldestReport				:BOOL;
	bCreate_ProcessReport				:BOOL;
	bCreate_SPReport					:BOOL;
END_STRUCT
END_TYPE

// ---- DUTs/ST_RX_Python.TcDUT
TYPE ST_RX_Python :
STRUCT
	stAuditExport				:ST_PythonHandshake;
	stSendReport				:ST_PythonHandshake;
	stBatchReport				:ST_PythonHandshake;
	stSP_BatchReport			:ST_PythonHandshake;
	stDiskCapacity				:ST_PythonHandshake;
	sDiskFree					:STRING(255);
	sDisckCapacity				:STRING(255);
END_STRUCT
END_TYPE

// ---- DUTs/ST_SeqControl.TcDUT
TYPE ST_SeqControl :
STRUCT
	iRecipeType					:INT;
	iPhaseType					:INT;
	bPhaseEnabled				:BOOL;
	iCurrentPhase				:INT;
	iCurrentStep				:INT;
	iPreviousStep				:INT;
	iTotalSteps					:INT;
	iStepNumbers				:ARRAY[0..10] OF INT;
	sStepDescription			:ARRAY[0..10] OF STRING;
	sPhaseTime					:STRING;
END_STRUCT
END_TYPE

// ---- DUTs/ST_Settings.TcDUT
TYPE ST_Settings :
STRUCT
	iSP_WaterFillingMaxTime			:DINT;
END_STRUCT
END_TYPE

// ---- DUTs/ST_SP_ProcessCmd.TcDUT
TYPE ST_SP_ProcessCmd :
STRUCT
	rMixerSpeed				:REAL;
	bMixerStart				:BOOL;
	rHeaterTemperature		:REAL;
	bHeaterStart			:BOOL;
END_STRUCT
END_TYPE

// ---- DUTs/ST_ToHMI.TcDUT
TYPE ST_ToHMI :
STRUCT
	bRecipeProd_Busy			:BOOL;
	iRecipeProd_Number			:INT;
	bRecipeClean_Busy			:BOOL;
	iRecipeClean_Number			:INT;
	iRecipeVerified_Number		:INT;
	sRecipeVerified_Names		:ARRAY[0..49] OF STRING;
	sRecipeProdVerified_Names	:ARRAY[0..49] OF STRING;
	sReport_OpenPath			:STRING;
	
	sAudit_OpenPath				:STRING;
	sUserMan_OpenPath			:STRING;
	
	sUserLogged					:STRING;
	
	sBatchOpen					:STRING;
	bBatchOpen					:BOOL;
	
	stHeader					:ST_Header;
	stControlsEN				:ST_EnableControl;
	stPID						:ST_PID;
	stPrompts					:ST_Prompts;
	arrSeqControl				:ARRAY[0..20] OF ST_SeqControl;
	rPhaseActiveTime			:REAL;
	sPhaseActiveTime			:STRING;
	bPhaseActiveTime_VIS		:BOOL;
	sLidOpenDelay				:STRING;
	bToolOperationReq			:BOOL;
	bAlarmDisabled				:BOOL;
	
	stSP						:ST_SP;
	
END_STRUCT
END_TYPE

// ---- DUTs/ST_toHMI/ST_EnableControl.TcDUT
TYPE ST_EnableControl :
STRUCT
	
	bLocalization_Img		:BOOL;
	bScreenShot_Img			:BOOL;

	bBatchEdit_Button		:BOOL;
	bBatchCreate_Button		:BOOL;
	
	bStop_Button			:BOOL;
	bPause_Button			:BOOL;
	bStart_Button			:BOOL;
	bAuto_Button			:BOOL;
	bService_Button			:BOOL;
	
	bOutlet_Buttons			:BOOL;
	bLid_Buttons			:BOOL;
	bSeal_Buttons			:BOOL;
	bTool_Buttons			:BOOL;
	bFindPos_Button			:BOOL;
	bTool_Container			:BOOL;
	
	bPump_Button			:BOOL;
	bMixer_Button			:BOOL;
	bSieve_Button			:BOOL;
	
	
END_STRUCT
END_TYPE

// ---- DUTs/ST_toHMI/ST_Header.TcDUT
TYPE ST_Header :
STRUCT
	iMachineMode				:INT; //0-Auto,1-Service
	iMachineStatus				:INT; //0-Stopped,1-Starting,2-Running,3-Stopping
	iBatchStatus				:INT;
	sActiveRecipe				:STRING;
	iCurrentPhaseName			:INT;
	iCurrentPhaseNo				:INT;
	iTotalPhaseNo				:INT;
	sBatchTime					:STRING;
	sPhaseTime					:STRING;
END_STRUCT
END_TYPE

// ---- DUTs/ST_toHMI/ST_PID.TcDUT
TYPE ST_PID :
STRUCT
	bShow_Labels				:BOOL;
	bHide_Buttons				:BOOL;	

	bFeeding					:BOOL;
	
	iMainUnit					:INT;
	
	iLid						:INT;
	iOutlet						:INT;
	iSieveSeal					:INT;
	iTool						:INT;
	iSieveMachine				:INT;
	
	iMixer						:INT;
	iChopper					:INT;
	
	
	iPAL_M882A					:INT;
	iPAL_M625					:INT;
	iPAL_M807					:INT;
	iFAL_M305A					:INT;
	iFAL_M205A					:INT;
	iFAL_M305C					:INT;
	iFAL_M205C					:INT;
	
	iSpray						:INT;
	
	iSieveSeal_Pipe				:INT;
	iPurgeSelect_Pipe			:INT;
	
	iSealChopper				:INT;
	iSealMixer					:INT;
	
	iMain_WIP_Pipe				:INT;
	iChopper_Pipe				:INT;
	iMixer_Pipe					:INT;
	
	iAspiration					:INT;
	iVacuum						:INT;
	iFilterClean				:INT;
	iCommonOutlet_Pipe			:INT;
	iDrain_Pipe					:INT;
	iOutletDrain_Pipe			:INT;
	iCommonDrain_Pipe			:INT;
	iSP_WIP_Pipe				:INT;
	iSP_WIP_Pipe2				:INT;
	iSPDrain_Pipe				:INT;
	iSP_Gran_Pipe				:INT;
	
	rWaterSimulation_Height		:REAL;
	rWaterSimulation_Top		:REAL;
	iWaterSimulation_Color		:INT;
	
	
	iEquipment					:INT;
	
END_STRUCT
END_TYPE

// ---- DUTs/ST_toHMI/ST_Prompts.TcDUT
TYPE ST_Prompts :
STRUCT
	bShow						:BOOL;
	bShow2						:BOOL;
	bBlink						:BOOL;
	iMessage					:INT;
END_STRUCT
END_TYPE

// ---- DUTs/ST_toHMI/ST_SP.TcDUT
TYPE ST_SP :
STRUCT
	iMachineStatus					:INT;
	sProcessTime					:STRING;
	sActiveProcessTime				:STRING;
	bAuto_EN						:BOOL;
	bService_EN						:BOOL;
	bStart_EN						:BOOL;
	bPause_EN						:BOOL;
	bStop_EN						:BOOL;
	bHeater_EN						:BOOL;
	bMixer_EN						:BOOL;
	bTime_EN						:BOOL;
	bRecipe_EN						:BOOL;
	bReportCreate_VIS				:BOOL;
END_STRUCT
END_TYPE

// ---- DUTs/ST_Trend.TcDUT
TYPE ST_Trend :
STRUCT
	rSP_Temperature_SP			:REAL;
	rSP_Temeprature_AP			:REAL;
	rSP_TemperatureW_AP			:REAL;
	rSP_MixingSpeed_SP			:REAL;
	rSP_MixingSpeed_AP			:REAL;
END_STRUCT
END_TYPE

// ---- DUTs/ST_TX_Python.TcDUT
TYPE ST_TX_Python :
STRUCT
	sAuditExportQuery				:STRING[300];
	sAuditFileName					:STRING[300];
	sBatchName						:STRING[300];
END_STRUCT
END_TYPE

// ---- GVLs/CONST.TcGVL
{attribute 'qualified_only'}
VAR_GLOBAL
	AMS_NETID					:STRING:='10.0.0.104.1.1';
	PROJECT_DIR					:STRING:='C:\TwinCAT\243401-ALDIO\';
	DB_ID						:UDINT:=1;
	ALARM_LOG_PATH				:STRING:='C:\TwinCAT\243401-ALDIO\Reports\1. Raw Data\AlarmLog.txt';
	STORE_REPORT_PATH			:STRING:='C:/TwinCAT/243401-ALDIO/Reports/2. Created/';
	DISK_CAPACITY				:STRING:='C:\\';
END_VAR

// ---- GVLs/GV.TcGVL
{attribute 'qualified_only'}
VAR_GLOBAL
	
	bWarning						:BOOL;
	bCritical						:BOOL;
	bDelete_DBs						:BOOL;
	stSeqControl					:ST_SeqControl;

	bUPSdetect						:BOOL;	
	bIPC_Overheated					:BOOL;

	sEmptyString					:STRING:='';
	
	//General
	stTime							:ST_Time;
	stHMI							:ST_HMI;
	stToHMI							:ST_ToHMI;
	stReport						:ST_Report;
	stProcessReport					:ST_Report;
	stAlarm							:ST_Alarm;
	stIPCDiag						:ST_Diagnostic;
	stTrend							:ST_Trend;
	

	stTX_Python						:ST_TX_Python;
	stRX_Python						:ST_RX_Python;
	
	stCleaningCmd					:ST_ProcessCmd;
	stProductionCmd					:ST_ProcessCmd;
	stAutoProcessCmd				:ST_ProcessCmd;
	stManProcessCmd					:ST_ProcessCmd2;
	stSPAutoProcessCmd				:ST_SP_ProcessCmd;
	

	
	bSP_BatchOpen					:BOOL;
	bSP_BatchClose					:BOOL;
	bAlarmOK						:BOOL;
	bSP_AlarmOK						:BOOL;
	
	iPP								:INT; //Current production process 
	iCP								:INT; //Current cleaning process
	iPrevPP							:INT; //Previous production process
	iPrevCP							:INT; //Previous cleaning process
	
		
	sProdPhases						:ARRAY[0..4] OF STRING:=['Feeding', 'Mixing', 'Granulation', 'Discharging'];
	sCleanPhases					:ARRAY[0..6] OF STRING:=['Pre-Cleaning', 'Main Cleaning', 'Rinsing', 'PW Cleaning',
														 'Draining', 'Blowing-out', 'Control'];
	arrPhaseEndpoint				:ARRAY[0..2] OF STRING:=['Auto', 'Manual', 'Mixer current'];
	arrChopper						:ARRAY[0..2] OF STRING:=['Off', 'Slow', 'Fast'];
	arrMedium						:ARRAY[0..1] OF STRING:=['Cold', 'Warm'];
	arrDetergent					:ARRAY[0..1] OF STRING:=['Off', 'On'];
	

	//Process variables
	rMixer_ActualSpeed				:REAL;
	rMixer_ActualCurrent			:REAL;
	rSieve_ActualSpeed				:REAL;
	rChopper_ActualCurrent			:REAL;
	
	rSP_Mixer_ActualSpeed			:REAL;
	rSP_ActualPressure				:REAL;
	rSP_Water_ActualTemperature		:REAL;
	rSP_Liquid_ActualTemperature	:REAL;
END_VAR
VAR_GLOBAL PERSISTENT
	sUserLogged						:STRING;	
	sGroupLogged					:STRING;
	
	bBatchOpen						:BOOL;
	bBatchClose						:BOOL;
	bBatchBusy						:BOOL;
	iRecipeType						:INT;
	stBatches						:ARRAY[0..9] OF ST_Batch;

	stControl						:ST_Control;
	stSP_Control					:ST_Control;
	stSettings						:ST_Settings;

	stBatch							:ST_Batch;
	stSP_Batch						:ST_Batch;
	stLastBatch						:ST_Batch;
END_VAR

// ---- GVLs/IN.TcGVL
{attribute 'qualified_only'}
VAR_GLOBAL PERSISTENT
	
	//DI1
	bFuseControlAC_OK						:BOOL:=TRUE;
	bFuseControlDC_NOK						:BOOL;
	bVoltageMonitor_NOK						:BOOL;
	bTemperatureCabinetPC_NOK				:BOOL;
	bTemperatureCabinetPLC_NOK				:BOOL;
	bCabinetFanMotorProtection_Trip			:BOOL;
	bEEXModules_OK							:BOOL:=TRUE;
	bEStop_Relay_OK							:BOOL:=TRUE;
	
	bEStop_Cabinet_NOK						:BOOL;
	bEStop_Operation_NOK					:BOOL;
	bCompressedAir_PAL882A_OK				:BOOL:=TRUE; 
	bCompressedAirWIP_PAL807_OK				:BOOL:=TRUE;
	bCompressedAirSeal_PAL625_OK			:BOOL:=TRUE;
	bLid_Closed								:BOOL;
	bOutletCleaningPos_Open					:BOOL; //Sto tocno e ova?
	bSieveMachine_InPos						:BOOL:=TRUE;
	
	//DI2
	bMixerThermalProtection_Fault			:BOOL;
	bChopperThermalProtection_Fault			:BOOL;
	bSieveThermalProtection_Fault			:BOOL;
	bMixerContactor_ON						:BOOL;
	bChopperContactor_ON					:BOOL;
	bSieveContactor_ON						:BOOL;
	bVacuumMP_Trip							:BOOL;
	bVacuumContactor_ON						:BOOL;
	
	bMixerTempOil_Trip						:BOOL;
	bMixerFrequency_Ready					:BOOL;
	bMixerFrequency_Run						:BOOL;
	bSieveFrequency_Ready					:BOOL;
	bSieveFrequency_Run						:BOOL;
	//DI3
	bFlowSealDrive_FAL205A_OK				:BOOL;
	bFlowSealChopper_FAL305A_OK				:BOOL;
	bFlowSealDrive_FAL205C_OK				:BOOL;
	bFlowSealChopper_FAL305C_OK				:BOOL;
	
	bOutletPos_Opened						:BOOL;
	bOutletPos_Closed						:BOOL;
	bToolPos_Down1							:BOOL:=TRUE;
	bToolPos_Down2							:BOOL:=TRUE;
	bToolPos_Up								:BOOL;
	bMixerTool_InPos						:BOOL;
	bLid_Open								:BOOL;
	
	//DI4
	bMixerStop_Button						:BOOL;
	bMixerStart_Button						:BOOL;
	bOutletOpen_Button						:BOOL;
	bOutletClose_Button						:BOOL;
	bSieveStop_Button						:BOOL;
	bSieveStart_Button						:BOOL;
	bVacuumStop_Button						:BOOL; 
	bVacuumStart_Button						:BOOL;
	
	bSP_Lid_Closed							:BOOL;
	bSP_Water_MinLevel						:BOOL;
	bSP_MixerFreq_Run						:BOOL;

	//TI1
	iSP_LiquidTemperature					:INT;
	iSP_VesselTemperature					:INT;
	// AI1
	iMixer_ActualSpeed						:INT;
	iMixer_ActualCurrent					:INT;
	iSieve_ActualSpeed						:INT;
	iChopper_ActualCurrent					:INT;
	//AI2
	iSP_ActualPressure						:INT;
	iSP_ActualSpeed							:INT;

	bReserveEx								:BOOL; //?

END_VAR

// ---- GVLs/OUT.TcGVL
{attribute 'qualified_only'}
VAR_GLOBAL
	//DO1
	bMixerContactor_ON					:BOOL;
	bMixerFrequency_Start				:BOOL;
	bChopper_Slow						:BOOL;
	bChopper_Fast						:BOOL;
	bSieveContactor_ON					:BOOL;
	bSieveFrequency_Start				:BOOL;
	bVacuum_Start						:BOOL;
	
	bOutlet_Valve_Open					:BOOL;
	bOutlet_Valve_Close					:BOOL;
	bTool_Valve_Lift					:BOOL;
	bTool_Valve_Lower					:BOOL;
	bLid_Valve_Close					:BOOL;
	bLid_Valve_Open						:BOOL;
	bSelSeave_On						:BOOL;
	bSelSeave_Off						:BOOL;
	
	//DO2
	bAirPurgeMax_V205A_V305A_1			:BOOL;
	bAirPurgeMin_V205A_V305A_2			:BOOL;
	bAspiration_V817C					:BOOL;
	bVacuum_V866A						:BOOL;
	bFilterClean_V861B					:BOOL;
	bAirInput_V882C						:BOOL;  //Glaven dovod za pnevmatikata, koga se vklucuva?
	bMixer_Air_V807_4					:BOOL;
	bChopper_Air_V807_6					:BOOL;
	
	bVentilationOutlet_V625D			:BOOL; //Ova e povrzano so outlet flapot, koga se vklucuva?
	bCleanAir_WIP_V807_1				:BOOL;
	bPurifiedWater_WIP_V807_2			:BOOL;
	bWarmWater_WIP_V807_3				:BOOL;
	bColdWater_WIP_V807_4				:BOOL;
	bDrain_WIP_V807_2					:BOOL;
	bMixer_WIP_V807_3					:BOOL;
	bChopper_WIP_V807_5					:BOOL;
	
	//DO3
	bSP_WIP								:BOOL;
	bSPDrain_WIP						:BOOL;
	bSP_Mixer_Start						:BOOL;
	bSP_Heater_ON						:BOOL;
	
	bMixerRun_Light						:BOOL;
	bOutletOpen_Light					:BOOL;
	bOutletClose_Light					:BOOL;
	bSieveRun_Light						:BOOL;
	bVacuumRun_Light						:BOOL;
	
	//AO1
	iMixerSpeed							:INT;
	iSieveSpeed							:INT;
	iSP_MixerSpeed						:INT;
END_VAR

// ---- GVLs/Recipes.TcGVL
{attribute 'qualified_only'}
VAR_GLOBAL
	Production						:ST_Recipe_Production;
	Cleaning						:ST_Recipe_Cleaning;

	Production_Empty				:ST_Recipe_Production;
	Cleaning_Empty					:ST_Recipe_Cleaning;
	
	Production_Phase_Empty			:ST_Production_Phases;
	Cleaning_Phase_Empty			:ST_Cleaning_Phases;
	
	Production_Phase_HMI			:ST_Production_Phases;
	Cleaning_Phase_HMI				:ST_Cleaning_Phases;
	Production_PhaseB_HMI			:ST_Production_Phases;
	Cleaning_PhaseB_HMI				:ST_Cleaning_Phases;
	
END_VAR
VAR_GLOBAL PERSISTENT
	Production_Active				:ST_Recipe_Production;
	Cleaning_Active					:ST_Recipe_Cleaning;
END_VAR

// ---- POUs/MAIN.TcPOU
PROGRAM MAIN
VAR
	bFirstCycle				:BOOL:=TRUE;
	tonFirstCycleDelay		:TON;
	bFirstCycleDelay		:BOOL;
	
	//UPS
	fbUPS					:FB_S_UPS_BAPI;
	eGlobalSUpsState 		:E_S_UPS_State;
	fbWritePersistent		:WritePersistentData;
	

	//IPC diagnostic
	fbReg					:FB_IPCDiag_Register;
	fbIPC_Temp				:FB_IPCDiag_ReadParameter;
	fbIPC_BootCnt			:FB_IPCDiag_ReadParameter;
	fbIPC_OperTime			:FB_IPCDiag_ReadParameter;	
	
	//Close application	
	fbCloseHMI				:NT_StartProcess;
	fbCloseRDP				:NT_StartProcess;
END_VAR

IF bFirstCycle THEN
	bFirstCycleDelay:=TRUE;
END_IF

tonFirstCycleDelay(IN:=bFirstCycleDelay,PT:=T#500MS);
IF tonFirstCycleDelay.Q THEN
	bFirstCycleDelay:=FALSE;
END_IF

P02_GlobalSystemTime();
P03_DiskSize();
P04_Screenshot();

P0_00_MAIN();
P1_00_MAIN();
P2_00_MAIN();
P3_00_MAIN();
P5_00_MAIN();

SIMULATION();

//Reset first cycle bit after reading all programs
bFirstCycle:=FALSE;

//********************DETECT UPS FAILURE*************************
fbUPS(sNetID:=CONST.AMS_NETID,
	iPLCPort:=851,
	tTimeout:=DEFAULT_ADS_TIMEOUT,
	eUpsMode:=eSUPS_WrPersistData_NoShutdown,
	ePersistentMode:=SPDM_2PASS,
	tRecoverTime:=T#10S,
	bPowerFailDetect=>GV.bUPSdetect, eState=>eGlobalSUpsState);

fbWritePersistent(NETID:=CONST.AMS_NETID,
	PORT:=851,
	START:=GV.stTime.bClock_60s,
	TMOUT:=T#10S);

//********************IPC DIAGNOSTIC*************************
fbReg(bExecute:=GV.stTime.bClock_5s,
	sNetId:=CONST.AMS_NETID);

//Motherboard temperature
fbIPC_Temp(bExecute:=fbReg.bValid,
	eParameterKey:=E_IPCDiag_ParameterKey.MB_Temperature,
	sNetId:=CONST.AMS_NETID,
	fbRegister:=fbReg);
IF NOT fbIPC_Temp.bBusy AND fbIPC_Temp.bValid THEN
	fbIPC_Temp.GetParameter(pBuffer:=ADR(GV.stIPCDiag.Temperature),
					nBufferSize:=SIZEOF(GV.stIPCDiag.Temperature));
END_IF

GV.bIPC_Overheated:= GV.stIPCDiag.Temperature > 80;
//Boot count
fbIPC_BootCnt(bExecute:=fbReg.bValid,
	eParameterKey:=E_IPCDiag_ParameterKey.MB_BootCnt,
	sNetId:=CONST.AMS_NETID,
	fbRegister:=fbReg);
IF NOT fbIPC_BootCnt.bBusy AND fbIPC_BootCnt.bValid THEN
	fbIPC_BootCnt.GetParameter(pBuffer:=ADR(GV.stIPCDiag.BootCount),
					nBufferSize:=SIZEOF(GV.stIPCDiag.BootCount));
END_IF
//Operation time
fbIPC_OperTime(bExecute:=fbReg.bValid,
	eParameterKey:=E_IPCDiag_ParameterKey.MB_OperationTime,
	sNetId:=CONST.AMS_NETID,
	fbRegister:=fbReg);
IF NOT fbIPC_OperTime.bBusy AND fbIPC_OperTime.bValid THEN
	fbIPC_OperTime.GetParameter(pBuffer:=ADR(GV.stIPCDiag.OperationTime),
					nBufferSize:=SIZEOF(GV.stIPCDiag.OperationTime));
END_IF


GV.stIPCDiag.OperationDuration:=F_OperationalTime(GV.stIPCDiag.OperationTime);


fbCloseHMI(NETID:='',
		PATHSTR:='C:\Windows\System32\taskkill.exe',
		DIRNAME:='C:\Windows\System32',
		COMNDLINE:='/F /IM "msedge.exe"',
		START:=GV.stHMI.bCloseHMI,
		TMOUT:=T#3S);
fbCloseRDP(NETID:='',
		PATHSTR:='C:\Windows\System32\taskkill.exe',
		DIRNAME:='C:\Windows\System32',
		COMNDLINE:='/F /IM "mstsc.exe"',
		START:=GV.stHMI.bCloseHMI,
		TMOUT:=T#3S);
			
GV.stHMI.bCloseHMI:=FALSE;

END_PROGRAM

// ---- POUs/P02_GlobalSystemTime.TcPOU
PROGRAM P02_GlobalSystemTime
VAR
	fbGlobalTime 		:FB_SystemDateTIme;
	
END_VAR

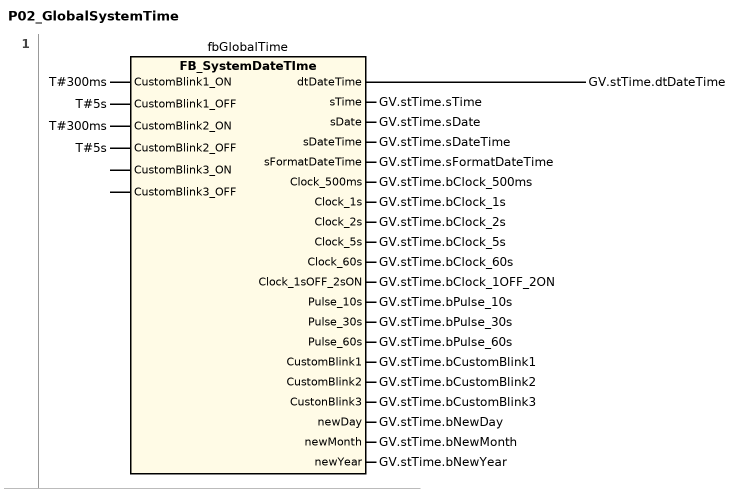
// NETWORK 1
fbGlobalTime(
    CustomBlink1_ON := T#300ms,
    CustomBlink1_OFF := T#5s,
    CustomBlink2_ON := T#300ms,
    CustomBlink2_OFF := T#5s,
    sTime => GV.stTime.sTime,
    sDate => GV.stTime.sDate,
    sDateTime => GV.stTime.sDateTime,
    sFormatDateTime => GV.stTime.sFormatDateTime,
    Clock_500ms => GV.stTime.bClock_500ms,
    Clock_1s => GV.stTime.bClock_1s,
    Clock_2s => GV.stTime.bClock_2s,
    Clock_5s => GV.stTime.bClock_5s,
    Clock_60s => GV.stTime.bClock_60s,
    Clock_1sOFF_2sON => GV.stTime.bClock_1OFF_2ON,
    Pulse_10s => GV.stTime.bPulse_10s,
    Pulse_30s => GV.stTime.bPulse_30s,
    Pulse_60s => GV.stTime.bPulse_60s,
    CustomBlink1 => GV.stTime.bCustomBlink1,
    CustomBlink2 => GV.stTime.bCustomBlink2,
    CustonBlink3 => GV.stTime.bCustomBlink3,
    newDay => GV.stTime.bNewDay,
    newMonth => GV.stTime.bNewMonth,
    newYear => GV.stTime.bNewYear); // FB_SystemDateTIme
GV.stTime.dtDateTime := fbGlobalTime.dtDateTime;

END_PROGRAM

// ---- FBs/FB_SystemDateTime.TcPOU
// Created by Dimitar Stojanov 06.2023 
// Install TC2_Utilities and Import ST_Time structure for fully functionality of this block


FUNCTION_BLOCK FB_SystemDateTime
VAR_INPUT
	CustomBlink1_ON		:TIME;
	CustomBlink1_OFF	:TIME;
	CustomBlink2_ON		:TIME;
	CustomBlink2_OFF	:TIME;
	CustomBlink3_ON		:TIME;
	CustomBlink3_OFF	:TIME;
END_VAR
VAR_OUTPUT
	dtDateTime		:DT;
	sTime			:STRING;
	sDate			:STRING;
	sDateTime		:STRING;
	sFormatDateTime	:STRING;
	Clock_500ms		:BOOL;
	Clock_1s		:BOOL;
	Clock_2s		:BOOL;
	Clock_5s		:BOOL;
	Clock_60s		:BOOL;
	Clock_1sOFF_2sON	:BOOL;
	Pulse_10s		:BOOL;
	Pulse_30s		:BOOL;
	Pulse_60s		:BOOL;
	CustomBlink1	:BOOL;
	CustomBlink2	:BOOL;
	CustonBlink3	:BOOL;
	newDay			:BOOL;
	newMonth		:BOOL;
	newYear			:BOOL;
END_VAR
VAR
	bFirstCycle		:BOOL:=TRUE;	

	fbTime			:FB_LocalSystemTime;
	systemDateTime	:TIMESTRUCT;
	
	Second			:STRING;
	Minute			:STRING;
	Hour			:STRING;
	Day				:STRING;
	Month			:STRING;
	Year			:STRING;
	
	iClock1s		:INT;
	TON_0: TON;
	TOF_0: TOF;
	TON_1: TON;
	TOF_1: TOF;
	TOF_2: TOF;
	TON_2: TON;
	TON_3: TON;
	TOF_3: TOF;
	TOF_4: TOF;
	TON_4: TON;
	TON_5: TON;
	TOF_5: TOF;
	TON_6: TON;
	TOF_6: TOF;
	TON_7: TON;
	TOF_7: TOF;
	TON_8: TON;
	TOF_8: TOF;
	
	TON_9: TON;
	TOF_9: TOF;
	TOF_10: TOF;
	TOF_11: TOF;
	TON_10: TON;
	TON_20: TON;
	TOF_20: TOF;
	TON_21: TON;
	TOF_21: TOF;
	TON_22: TON;
	TOF_22: TOF;
	
	bDelay			:BOOL;
	TON_DELAY		:TON;
END_VAR

VAR PERSISTENT
	CurrentDay		:WORD;
	CurrentMonth	:WORD;
	CurrentYear		:WORD;
END_VAR

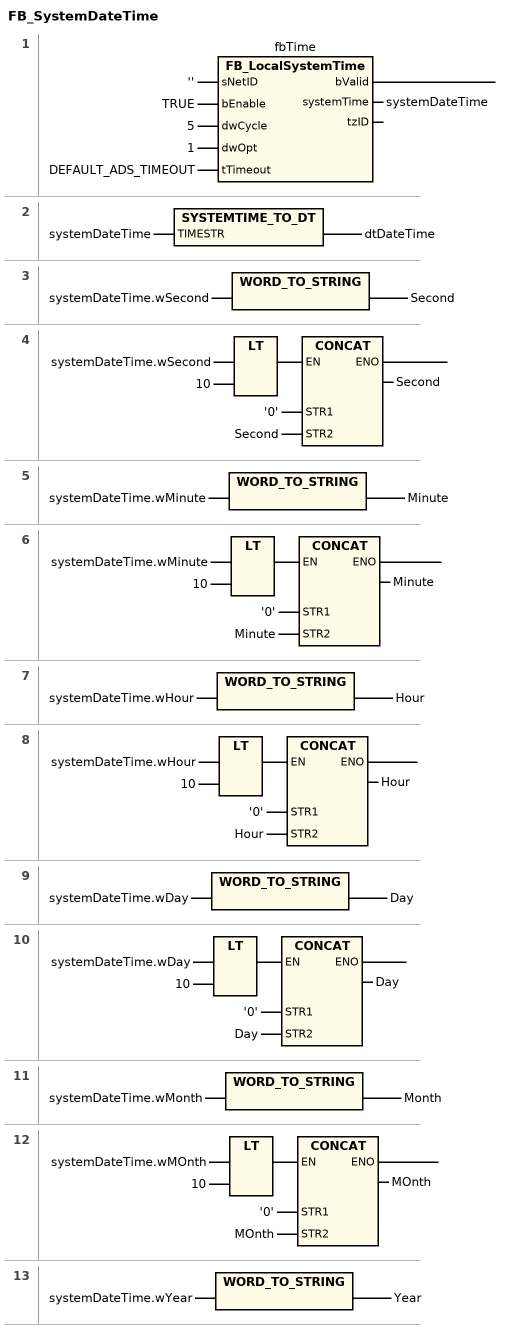
// NETWORK 1
fbTime(
    sNetID := '',
    bEnable := TRUE,
    dwCycle := 5,
    dwOpt := 1,
    tTimeout := DEFAULT_ADS_TIMEOUT,
    systemTime => systemDateTime); // FB_LocalSystemTime

// NETWORK 2
dtDateTime := SYSTEMTIME_TO_DT(TIMESTR := systemDateTime);

// NETWORK 3
Second := WORD_TO_STRING(systemDateTime.wSecond);

// NETWORK 4
IF systemDateTime.wSecond < 10 THEN Second := CONCAT(STR1 := '0', STR2 := Second); END_IF

// NETWORK 5
Minute := WORD_TO_STRING(systemDateTime.wMinute);

// NETWORK 6
IF systemDateTime.wMinute < 10 THEN Minute := CONCAT(STR1 := '0', STR2 := Minute); END_IF

// NETWORK 7
Hour := WORD_TO_STRING(systemDateTime.wHour);

// NETWORK 8
IF systemDateTime.wHour < 10 THEN Hour := CONCAT(STR1 := '0', STR2 := Hour); END_IF

// NETWORK 9
Day := WORD_TO_STRING(systemDateTime.wDay);

// NETWORK 10
IF systemDateTime.wDay < 10 THEN Day := CONCAT(STR1 := '0', STR2 := Day); END_IF

// NETWORK 11
Month := WORD_TO_STRING(systemDateTime.wMonth);

// NETWORK 12
IF systemDateTime.wMOnth < 10 THEN MOnth := CONCAT(STR1 := '0', STR2 := MOnth); END_IF

// NETWORK 13
Year := WORD_TO_STRING(systemDateTime.wYear);

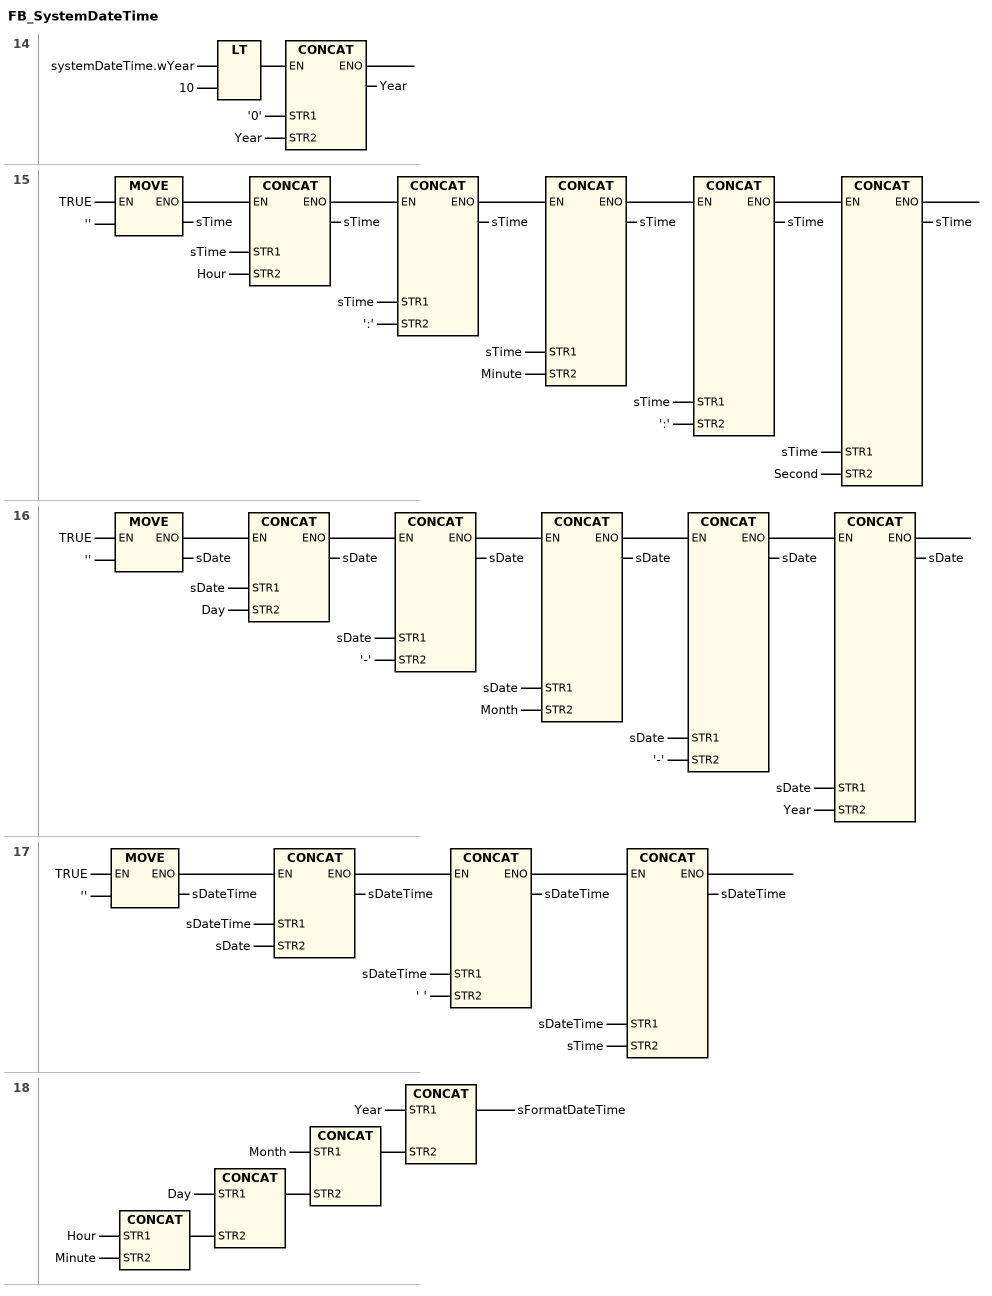
// NETWORK 14
IF systemDateTime.wYear < 10 THEN Year := CONCAT(STR1 := '0', STR2 := Year); END_IF

// NETWORK 15
sTime := '';
sTime := CONCAT(STR1 := sTime, STR2 := Hour);
sTime := CONCAT(STR1 := sTime, STR2 := ':');
sTime := CONCAT(STR1 := sTime, STR2 := Minute);
sTime := CONCAT(STR1 := sTime, STR2 := ':');
sTime := CONCAT(STR1 := sTime, STR2 := Second);

// NETWORK 16
sDate := '';
sDate := CONCAT(STR1 := sDate, STR2 := Day);
sDate := CONCAT(STR1 := sDate, STR2 := '-');
sDate := CONCAT(STR1 := sDate, STR2 := Month);
sDate := CONCAT(STR1 := sDate, STR2 := '-');
sDate := CONCAT(STR1 := sDate, STR2 := Year);

// NETWORK 17
sDateTime := '';
sDateTime := CONCAT(STR1 := sDateTime, STR2 := sDate);
sDateTime := CONCAT(STR1 := sDateTime, STR2 := ' ');
sDateTime := CONCAT(STR1 := sDateTime, STR2 := sTime);

// NETWORK 18
sFormatDateTime := CONCAT(STR1 := Year, STR2 := CONCAT(STR1 := Month, STR2 := CONCAT(STR1 := Day, STR2 := CONCAT(STR1 := Hour, STR2 := Minute))));

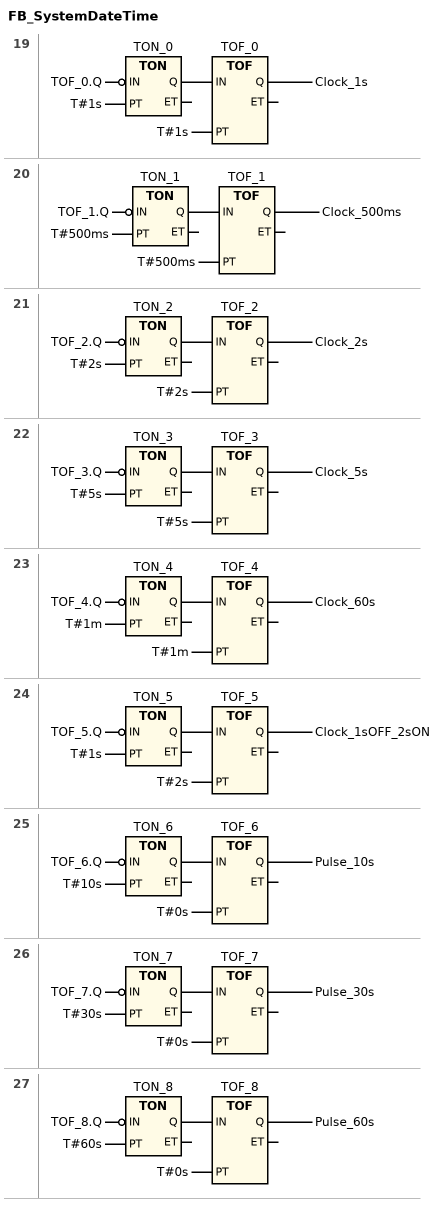
// NETWORK 19
TON_0(IN := NOT TOF_0.Q, PT := T#1s); // TON
TOF_0(IN := TON_0.Q, PT := T#1s); // TOF
Clock_1s := TOF_0.Q;

// NETWORK 20
TON_1(IN := NOT TOF_1.Q, PT := T#500ms); // TON
TOF_1(IN := TON_1.Q, PT := T#500ms); // TOF
Clock_500ms := TOF_1.Q;

// NETWORK 21
TON_2(IN := NOT TOF_2.Q, PT := T#2s); // TON
TOF_2(IN := TON_2.Q, PT := T#2s); // TOF
Clock_2s := TOF_2.Q;

// NETWORK 22
TON_3(IN := NOT TOF_3.Q, PT := T#5s); // TON
TOF_3(IN := TON_3.Q, PT := T#5s); // TOF
Clock_5s := TOF_3.Q;

// NETWORK 23
TON_4(IN := NOT TOF_4.Q, PT := T#1m); // TON
TOF_4(IN := TON_4.Q, PT := T#1m); // TOF
Clock_60s := TOF_4.Q;

// NETWORK 24
TON_5(IN := NOT TOF_5.Q, PT := T#1s); // TON
TOF_5(IN := TON_5.Q, PT := T#2s); // TOF
Clock_1sOFF_2sON := TOF_5.Q;

// NETWORK 25
TON_6(IN := NOT TOF_6.Q, PT := T#10s); // TON
TOF_6(IN := TON_6.Q, PT := T#0s); // TOF
Pulse_10s := TOF_6.Q;

// NETWORK 26
TON_7(IN := NOT TOF_7.Q, PT := T#30s); // TON
TOF_7(IN := TON_7.Q, PT := T#0s); // TOF
Pulse_30s := TOF_7.Q;

// NETWORK 27
TON_8(IN := NOT TOF_8.Q, PT := T#60s); // TON
TOF_8(IN := TON_8.Q, PT := T#0s); // TOF
Pulse_60s := TOF_8.Q;

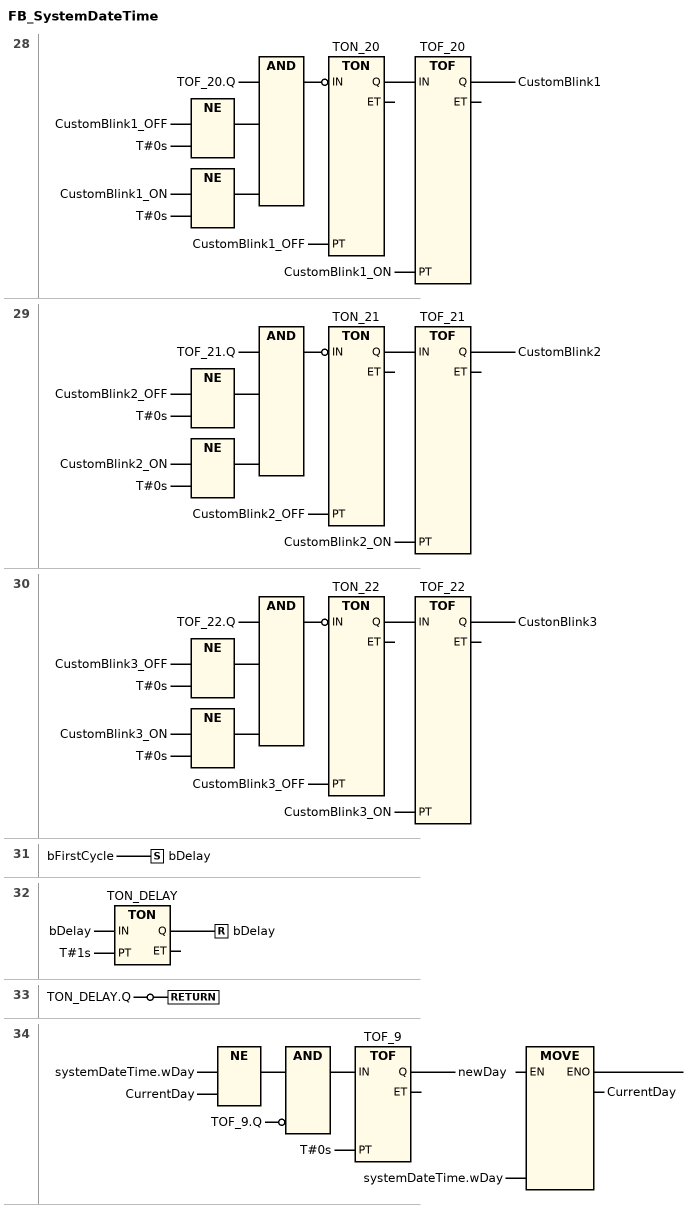
// NETWORK 28
TON_20(IN := NOT (TOF_20.Q AND CustomBlink1_OFF <> T#0s AND CustomBlink1_ON <> T#0s), PT := CustomBlink1_OFF); // TON
TOF_20(IN := TON_20.Q, PT := CustomBlink1_ON); // TOF
CustomBlink1 := TOF_20.Q;

// NETWORK 29
TON_21(IN := NOT (TOF_21.Q AND CustomBlink2_OFF <> T#0s AND CustomBlink2_ON <> T#0s), PT := CustomBlink2_OFF); // TON
TOF_21(IN := TON_21.Q, PT := CustomBlink2_ON); // TOF
CustomBlink2 := TOF_21.Q;

// NETWORK 30
TON_22(IN := NOT (TOF_22.Q AND CustomBlink3_OFF <> T#0s AND CustomBlink3_ON <> T#0s), PT := CustomBlink3_OFF); // TON
TOF_22(IN := TON_22.Q, PT := CustomBlink3_ON); // TOF
CustonBlink3 := TOF_22.Q;

// NETWORK 31
bDelay S= bFirstCycle;

// NETWORK 32
TON_DELAY(IN := bDelay, PT := T#1s); // TON
bDelay R= TON_DELAY.Q;

// NETWORK 33
IF NOT TON_DELAY.Q THEN RETURN; END_IF

// NETWORK 34
TOF_9(IN := systemDateTime.wDay <> CurrentDay AND NOT TOF_9.Q, PT := T#0s); // TOF
newDay := TOF_9.Q;
IF TOF_9.Q THEN CurrentDay := systemDateTime.wDay; END_IF

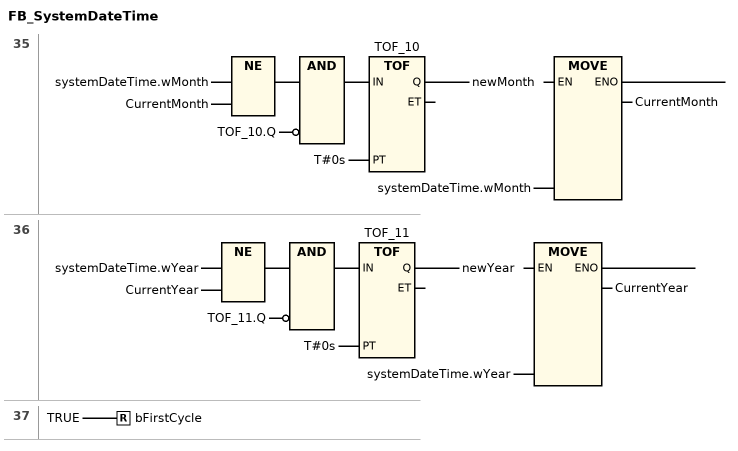
// NETWORK 35
TOF_10(IN := systemDateTime.wMonth <> CurrentMonth AND NOT TOF_10.Q, PT := T#0s); // TOF
newMonth := TOF_10.Q;
IF TOF_10.Q THEN CurrentMonth := systemDateTime.wMonth; END_IF

// NETWORK 36
TOF_11(IN := systemDateTime.wYear <> CurrentYear AND NOT TOF_11.Q, PT := T#0s); // TOF
newYear := TOF_11.Q;
IF TOF_11.Q THEN CurrentYear := systemDateTime.wYear; END_IF

// NETWORK 37
bFirstCycle R= TRUE;

END_FUNCTION_BLOCK

// ---- POUs/P03_DiskSize.TcPOU
PROGRAM P03_DiskSize
VAR
	fbSize						:FB_PythonScript;
	bReadAfterPowerUp			:BOOL;
	tonReadAfterPowerUpDelay	:TON;
END_VAR

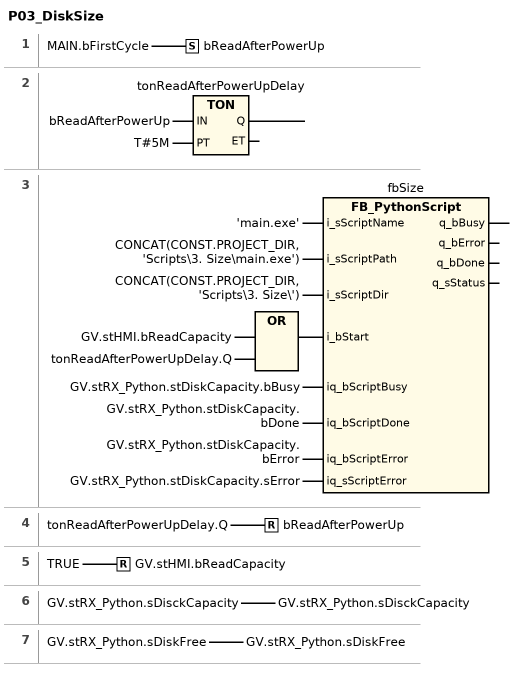
// NETWORK 1
bReadAfterPowerUp S= MAIN.bFirstCycle;

// NETWORK 2
tonReadAfterPowerUpDelay(IN := bReadAfterPowerUp, PT := T#5M); // TON

// NETWORK 3
fbSize(
    i_sScriptName := 'main.exe',
    i_sScriptPath := CONCAT(CONST.PROJECT_DIR,'Scripts\3. Size\main.exe'),
    i_sScriptDir := CONCAT(CONST.PROJECT_DIR,'Scripts\3. Size\'),
    i_bStart := GV.stHMI.bReadCapacity OR tonReadAfterPowerUpDelay.Q,
    iq_bScriptBusy := GV.stRX_Python.stDiskCapacity.bBusy,
    iq_bScriptDone := GV.stRX_Python.stDiskCapacity.bDone,
    iq_bScriptError := GV.stRX_Python.stDiskCapacity.bError,
    iq_sScriptError := GV.stRX_Python.stDiskCapacity.sError); // FB_PythonScript

// NETWORK 4
bReadAfterPowerUp R= tonReadAfterPowerUpDelay.Q;

// NETWORK 5
GV.stHMI.bReadCapacity R= TRUE;

// NETWORK 6
GV.stRX_Python.sDisckCapacity := GV.stRX_Python.sDisckCapacity;

// NETWORK 7
GV.stRX_Python.sDiskFree := GV.stRX_Python.sDiskFree;

END_PROGRAM

// ---- FBs/FB_PythonScript.TcPOU
FUNCTION_BLOCK FB_PythonScript
VAR_INPUT
	i_sScriptName		:STRING;
	i_sScriptPath		:STRING;
	i_sScriptDir		:STRING;
	i_bStart			:BOOL;
END_VAR
VAR_IN_OUT
	iq_bScriptBusy		:BOOL;
	iq_bScriptDone		:BOOL;
	iq_bScriptError		:BOOL;
	iq_sScriptError		:STRING;
END_VAR
VAR_OUTPUT
	q_bBusy				:BOOL;
	q_bError			:BOOL;
	q_bDone				:BOOL;
	q_sStatus			:STRING;
END_VAR
VAR
	ntProcess			:NT_StartProcess;
	bStartNT			:BOOL;

	iStep				:INT;
	tTimeOut_TON1		:TON;
	tTimeOut1			:TIME;
	tTimeOut_TON2		:TON;
	tTimeOut2			:TIME;
END_VAR

ACT_StartProcess();

tTimeOut1:=T#300S;
tTimeOut2:=T#300S;

q_sStatus:=iq_sScriptError;

CASE iStep OF
	
	0:

		q_bBusy:=FALSE;
		tTimeOut_TON1(IN:=FALSE,PT:=tTimeOut1);
		tTimeOut_TON2(IN:=FALSE,PT:=tTimeOut2);
	
		IF i_bStart THEN
			q_bError:=FALSE;
			q_bDone:=FALSE;
			q_bBusy:=TRUE;
			
			iq_bScriptBusy:=FALSE;
			iq_bScriptDone:=FALSE;
			iq_bScriptError:=FALSE;
			iq_sScriptError:='';
			
			iStep:=10;
		END_IF
	
	10:
		bStartNT:=TRUE;
		IF ntProcess.BUSY THEN
			iStep:=15;
		END_IF
	
	15:
		IF NOT ntProcess.BUSY THEN
			iStep:=20;
		ELSIF ntProcess.ERR THEN
			iStep:=999;
		END_IF
	20:
		tTimeOut_TON1(IN:=TRUE,PT:=tTimeOut1);
		IF NOT iq_bScriptDone AND NOT iq_bScriptError THEN
			iStep:=30;
		ELSIF tTimeOut_TON1.Q OR iq_bScriptError THEN
			iStep:=999;
		END_IF
	30:
		tTimeOut_TON2(IN:=TRUE,PT:=tTimeOut2);
		IF iq_bScriptDone AND NOT iq_bScriptError THEN 
			iStep:=50;	
		ELSIF tTimeOut_TON2.Q OR iq_bScriptError THEN
			iStep:=999;
		END_IF
		
	50:
		q_bDone:=TRUE;
		iStep:=0;
	999:
		
		q_bError:=TRUE;
		iStep:=0;
		
		
END_CASE

ACTION ACT_StartProcess:
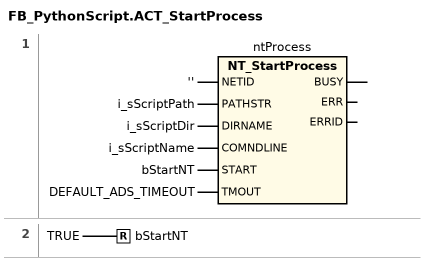
// NETWORK 1
ntProcess(
    NETID := '',
    PATHSTR := i_sScriptPath,
    DIRNAME := i_sScriptDir,
    COMNDLINE := i_sScriptName,
    START := bStartNT,
    TMOUT := DEFAULT_ADS_TIMEOUT); // NT_StartProcess

// NETWORK 2
bStartNT R= TRUE;
END_ACTION

END_FUNCTION_BLOCK

// ---- POUs/P04_Screenshot.TcPOU
PROGRAM P04_Screenshot
VAR
		fbScreenshot					:NT_StartProcess;
		tonDisable						:TON;
		bDisable						:BOOL;
END_VAR

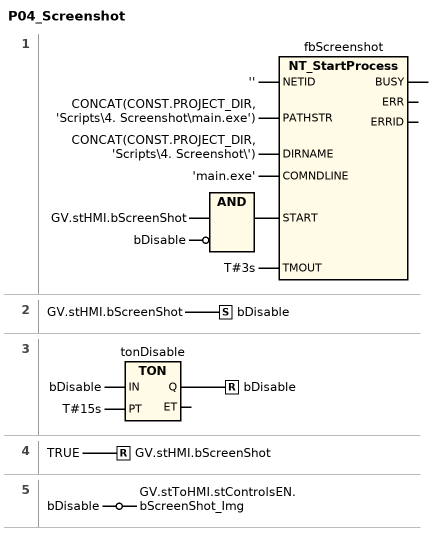
// NETWORK 1
fbScreenshot(
    NETID := '',
    PATHSTR := CONCAT(CONST.PROJECT_DIR,'Scripts\4. Screenshot\main.exe'),
    DIRNAME := CONCAT(CONST.PROJECT_DIR,'Scripts\4. Screenshot\'),
    COMNDLINE := 'main.exe',
    START := GV.stHMI.bScreenShot AND NOT bDisable,
    TMOUT := T#3s); // NT_StartProcess

// NETWORK 2
bDisable S= GV.stHMI.bScreenShot;

// NETWORK 3
tonDisable(IN := bDisable, PT := T#15s); // TON
bDisable R= tonDisable.Q;

// NETWORK 4
GV.stHMI.bScreenShot R= TRUE;

// NETWORK 5
GV.stToHMI.stControlsEN.bScreenShot_Img := NOT bDisable;

END_PROGRAM

// ---- POUs/0. Input/P0_00_MAIN.TcPOU
PROGRAM P0_00_MAIN
VAR
	test1: BOOL;
	test2: BOOL;
	test3: BOOL;
	test: BOOl;
END_VAR

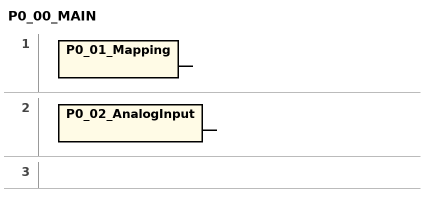
// NETWORK 1
P0_01_Mapping();

// NETWORK 2
P0_02_AnalogInput();

// NETWORK 3

END_PROGRAM

// ---- POUs/0. Input/P0_01_Mapping.TcPOU
PROGRAM P0_01_Mapping
VAR
	
	AI_SPARE								:INT;
	DI_SPARE								:BOOL;
	AO_SPARE								:INT:=0;
	DO_SPARE								:BOOL:=FALSE;

	AI1										:ST_EL3174;
	AI2										:ST_EL3174;
	DI1										:ST_EL1819;
	DI2										:ST_EL1819;
	DI3										:ST_EL1819;
	DI4										:ST_EL1819;
	PS										:ST_EL9110;
	AO1										:ST_EL4124;
	AO2										:ST_EL4124;
	DO1										:ST_EL2809;
	DO2										:ST_EL2809;
	DO3										:ST_EL2809;
	DO4										:ST_EL2809;
	
	bIO_Card_Failure						:BOOL;

END_VAR

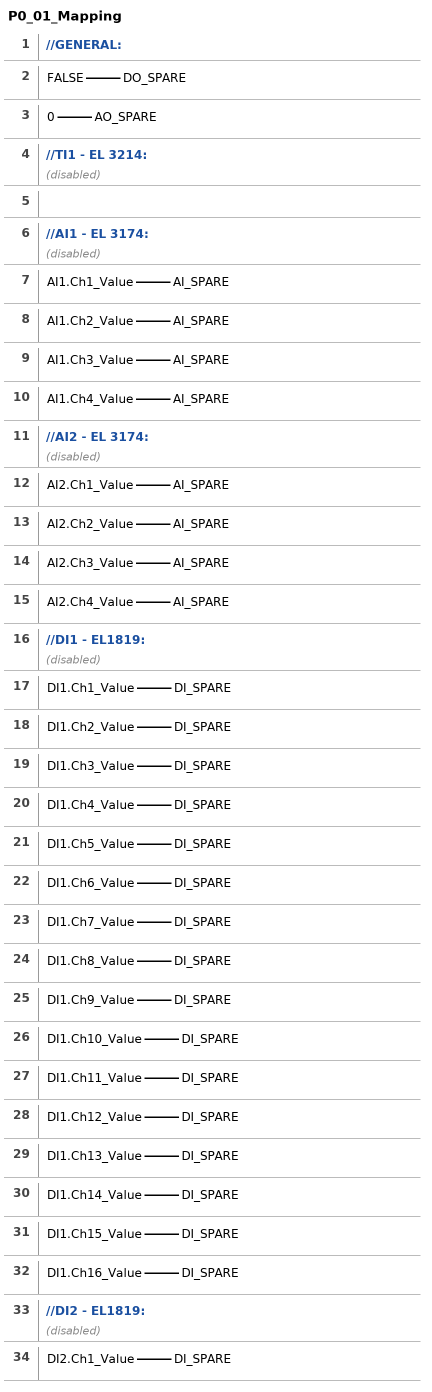
// NETWORK 1
// label: //GENERAL

// NETWORK 2
DO_SPARE := FALSE;

// NETWORK 3
AO_SPARE := 0;

// NETWORK 4 (disabled)
// label: //TI1 - EL 3214

// NETWORK 5

// NETWORK 6 (disabled)
// label: //AI1 - EL 3174

// NETWORK 7
AI_SPARE := AI1.Ch1_Value;

// NETWORK 8
AI_SPARE := AI1.Ch2_Value;

// NETWORK 9
AI_SPARE := AI1.Ch3_Value;

// NETWORK 10
AI_SPARE := AI1.Ch4_Value;

// NETWORK 11 (disabled)
// label: //AI2 - EL 3174

// NETWORK 12
AI_SPARE := AI2.Ch1_Value;

// NETWORK 13
AI_SPARE := AI2.Ch2_Value;

// NETWORK 14
AI_SPARE := AI2.Ch3_Value;

// NETWORK 15
AI_SPARE := AI2.Ch4_Value;

// NETWORK 16 (disabled)
// label: //DI1 - EL1819

// NETWORK 17
DI_SPARE := DI1.Ch1_Value;

// NETWORK 18
DI_SPARE := DI1.Ch2_Value;

// NETWORK 19
DI_SPARE := DI1.Ch3_Value;

// NETWORK 20
DI_SPARE := DI1.Ch4_Value;

// NETWORK 21
DI_SPARE := DI1.Ch5_Value;

// NETWORK 22
DI_SPARE := DI1.Ch6_Value;

// NETWORK 23
DI_SPARE := DI1.Ch7_Value;

// NETWORK 24
DI_SPARE := DI1.Ch8_Value;

// NETWORK 25
DI_SPARE := DI1.Ch9_Value;

// NETWORK 26
DI_SPARE := DI1.Ch10_Value;

// NETWORK 27
DI_SPARE := DI1.Ch11_Value;

// NETWORK 28
DI_SPARE := DI1.Ch12_Value;

// NETWORK 29
DI_SPARE := DI1.Ch13_Value;

// NETWORK 30
DI_SPARE := DI1.Ch14_Value;

// NETWORK 31
DI_SPARE := DI1.Ch15_Value;

// NETWORK 32
DI_SPARE := DI1.Ch16_Value;

// NETWORK 33 (disabled)
// label: //DI2 - EL1819

// NETWORK 34
DI_SPARE := DI2.Ch1_Value;

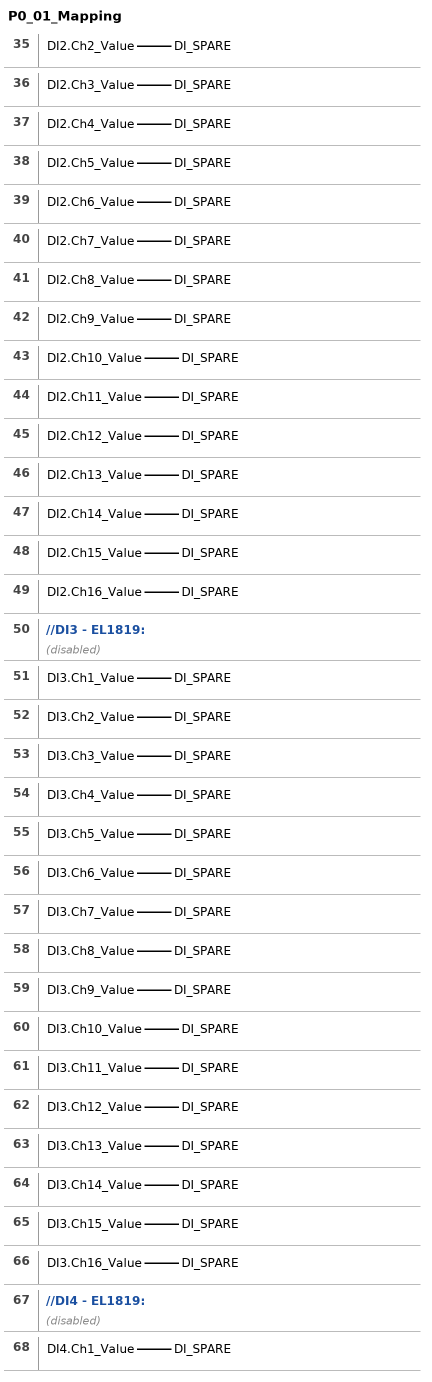
// NETWORK 35
DI_SPARE := DI2.Ch2_Value;

// NETWORK 36
DI_SPARE := DI2.Ch3_Value;

// NETWORK 37
DI_SPARE := DI2.Ch4_Value;

// NETWORK 38
DI_SPARE := DI2.Ch5_Value;

// NETWORK 39
DI_SPARE := DI2.Ch6_Value;

// NETWORK 40
DI_SPARE := DI2.Ch7_Value;

// NETWORK 41
DI_SPARE := DI2.Ch8_Value;

// NETWORK 42
DI_SPARE := DI2.Ch9_Value;

// NETWORK 43
DI_SPARE := DI2.Ch10_Value;

// NETWORK 44
DI_SPARE := DI2.Ch11_Value;

// NETWORK 45
DI_SPARE := DI2.Ch12_Value;

// NETWORK 46
DI_SPARE := DI2.Ch13_Value;

// NETWORK 47
DI_SPARE := DI2.Ch14_Value;

// NETWORK 48
DI_SPARE := DI2.Ch15_Value;

// NETWORK 49
DI_SPARE := DI2.Ch16_Value;

// NETWORK 50 (disabled)
// label: //DI3 - EL1819

// NETWORK 51
DI_SPARE := DI3.Ch1_Value;

// NETWORK 52
DI_SPARE := DI3.Ch2_Value;

// NETWORK 53
DI_SPARE := DI3.Ch3_Value;

// NETWORK 54
DI_SPARE := DI3.Ch4_Value;

// NETWORK 55
DI_SPARE := DI3.Ch5_Value;

// NETWORK 56
DI_SPARE := DI3.Ch6_Value;

// NETWORK 57
DI_SPARE := DI3.Ch7_Value;

// NETWORK 58
DI_SPARE := DI3.Ch8_Value;

// NETWORK 59
DI_SPARE := DI3.Ch9_Value;

// NETWORK 60
DI_SPARE := DI3.Ch10_Value;

// NETWORK 61
DI_SPARE := DI3.Ch11_Value;

// NETWORK 62
DI_SPARE := DI3.Ch12_Value;

// NETWORK 63
DI_SPARE := DI3.Ch13_Value;

// NETWORK 64
DI_SPARE := DI3.Ch14_Value;

// NETWORK 65
DI_SPARE := DI3.Ch15_Value;

// NETWORK 66
DI_SPARE := DI3.Ch16_Value;

// NETWORK 67 (disabled)
// label: //DI4 - EL1819

// NETWORK 68
DI_SPARE := DI4.Ch1_Value;

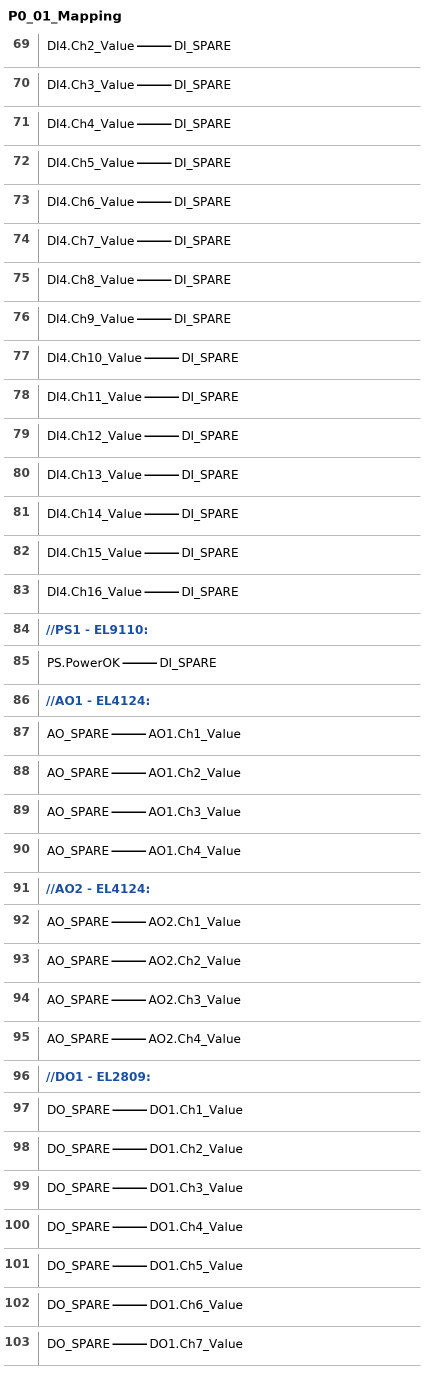
// NETWORK 69
DI_SPARE := DI4.Ch2_Value;

// NETWORK 70
DI_SPARE := DI4.Ch3_Value;

// NETWORK 71
DI_SPARE := DI4.Ch4_Value;

// NETWORK 72
DI_SPARE := DI4.Ch5_Value;

// NETWORK 73
DI_SPARE := DI4.Ch6_Value;

// NETWORK 74
DI_SPARE := DI4.Ch7_Value;

// NETWORK 75
DI_SPARE := DI4.Ch8_Value;

// NETWORK 76
DI_SPARE := DI4.Ch9_Value;

// NETWORK 77
DI_SPARE := DI4.Ch10_Value;

// NETWORK 78
DI_SPARE := DI4.Ch11_Value;

// NETWORK 79
DI_SPARE := DI4.Ch12_Value;

// NETWORK 80
DI_SPARE := DI4.Ch13_Value;

// NETWORK 81
DI_SPARE := DI4.Ch14_Value;

// NETWORK 82
DI_SPARE := DI4.Ch15_Value;

// NETWORK 83
DI_SPARE := DI4.Ch16_Value;

// NETWORK 84
// label: //PS1 - EL9110

// NETWORK 85
DI_SPARE := PS.PowerOK;

// NETWORK 86
// label: //AO1 - EL4124

// NETWORK 87
AO1.Ch1_Value := AO_SPARE;

// NETWORK 88
AO1.Ch2_Value := AO_SPARE;

// NETWORK 89
AO1.Ch3_Value := AO_SPARE;

// NETWORK 90
AO1.Ch4_Value := AO_SPARE;

// NETWORK 91
// label: //AO2 - EL4124

// NETWORK 92
AO2.Ch1_Value := AO_SPARE;

// NETWORK 93
AO2.Ch2_Value := AO_SPARE;

// NETWORK 94
AO2.Ch3_Value := AO_SPARE;

// NETWORK 95
AO2.Ch4_Value := AO_SPARE;

// NETWORK 96
// label: //DO1 - EL2809

// NETWORK 97
DO1.Ch1_Value := DO_SPARE;

// NETWORK 98
DO1.Ch2_Value := DO_SPARE;

// NETWORK 99
DO1.Ch3_Value := DO_SPARE;

// NETWORK 100
DO1.Ch4_Value := DO_SPARE;

// NETWORK 101
DO1.Ch5_Value := DO_SPARE;

// NETWORK 102
DO1.Ch6_Value := DO_SPARE;

// NETWORK 103
DO1.Ch7_Value := DO_SPARE;

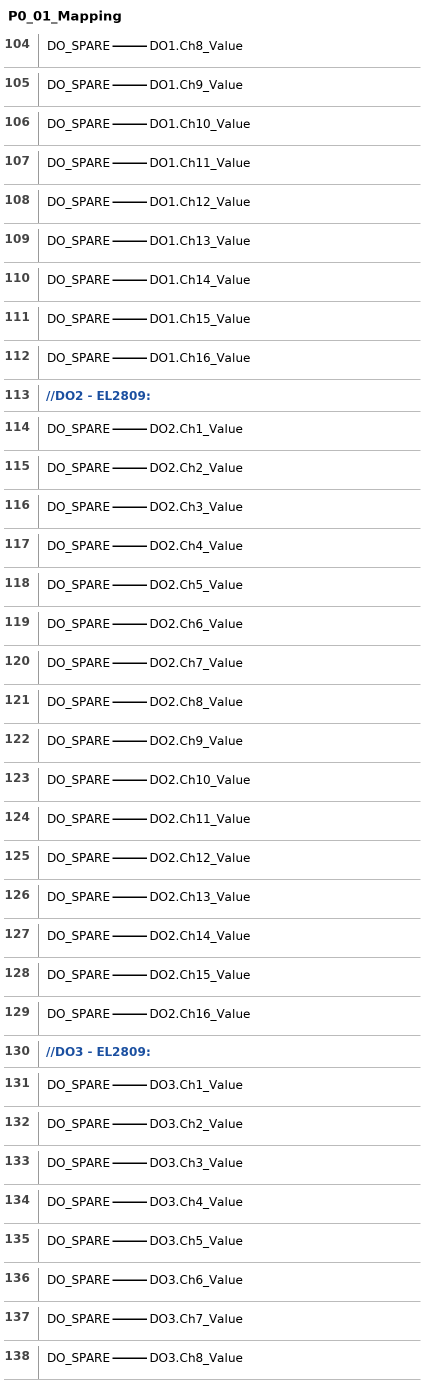
// NETWORK 104
DO1.Ch8_Value := DO_SPARE;

// NETWORK 105
DO1.Ch9_Value := DO_SPARE;

// NETWORK 106
DO1.Ch10_Value := DO_SPARE;

// NETWORK 107
DO1.Ch11_Value := DO_SPARE;

// NETWORK 108
DO1.Ch12_Value := DO_SPARE;

// NETWORK 109
DO1.Ch13_Value := DO_SPARE;

// NETWORK 110
DO1.Ch14_Value := DO_SPARE;

// NETWORK 111
DO1.Ch15_Value := DO_SPARE;

// NETWORK 112
DO1.Ch16_Value := DO_SPARE;

// NETWORK 113
// label: //DO2 - EL2809

// NETWORK 114
DO2.Ch1_Value := DO_SPARE;

// NETWORK 115
DO2.Ch2_Value := DO_SPARE;

// NETWORK 116
DO2.Ch3_Value := DO_SPARE;

// NETWORK 117
DO2.Ch4_Value := DO_SPARE;

// NETWORK 118
DO2.Ch5_Value := DO_SPARE;

// NETWORK 119
DO2.Ch6_Value := DO_SPARE;

// NETWORK 120
DO2.Ch7_Value := DO_SPARE;

// NETWORK 121
DO2.Ch8_Value := DO_SPARE;

// NETWORK 122
DO2.Ch9_Value := DO_SPARE;

// NETWORK 123
DO2.Ch10_Value := DO_SPARE;

// NETWORK 124
DO2.Ch11_Value := DO_SPARE;

// NETWORK 125
DO2.Ch12_Value := DO_SPARE;

// NETWORK 126
DO2.Ch13_Value := DO_SPARE;

// NETWORK 127
DO2.Ch14_Value := DO_SPARE;

// NETWORK 128
DO2.Ch15_Value := DO_SPARE;

// NETWORK 129
DO2.Ch16_Value := DO_SPARE;

// NETWORK 130
// label: //DO3 - EL2809

// NETWORK 131
DO3.Ch1_Value := DO_SPARE;

// NETWORK 132
DO3.Ch2_Value := DO_SPARE;

// NETWORK 133
DO3.Ch3_Value := DO_SPARE;

// NETWORK 134
DO3.Ch4_Value := DO_SPARE;

// NETWORK 135
DO3.Ch5_Value := DO_SPARE;

// NETWORK 136
DO3.Ch6_Value := DO_SPARE;

// NETWORK 137
DO3.Ch7_Value := DO_SPARE;

// NETWORK 138
DO3.Ch8_Value := DO_SPARE;

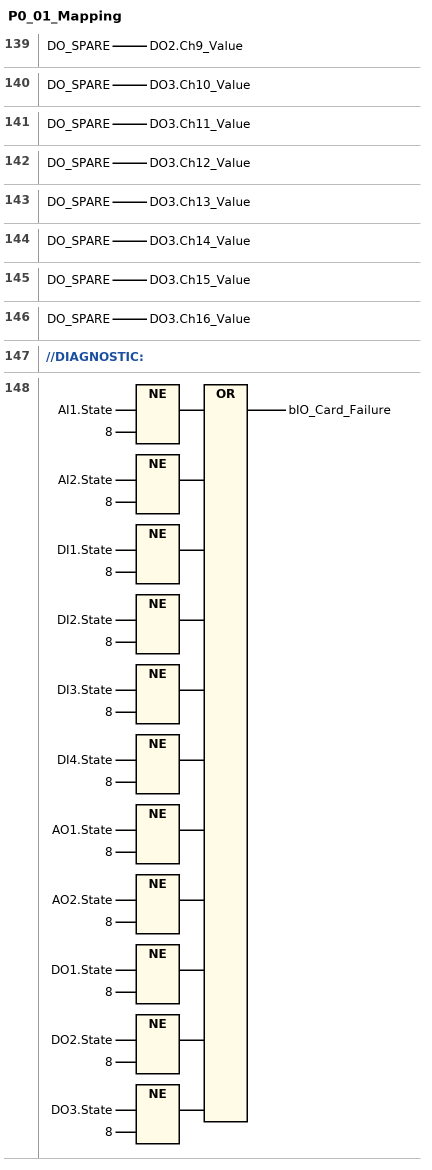
// NETWORK 139
DO2.Ch9_Value := DO_SPARE;

// NETWORK 140
DO3.Ch10_Value := DO_SPARE;

// NETWORK 141
DO3.Ch11_Value := DO_SPARE;

// NETWORK 142
DO3.Ch12_Value := DO_SPARE;

// NETWORK 143
DO3.Ch13_Value := DO_SPARE;

// NETWORK 144
DO3.Ch14_Value := DO_SPARE;

// NETWORK 145
DO3.Ch15_Value := DO_SPARE;

// NETWORK 146
DO3.Ch16_Value := DO_SPARE;

// NETWORK 147
// label: //DIAGNOSTIC

// NETWORK 148
bIO_Card_Failure := AI1.State <> 8 OR AI2.State <> 8 OR DI1.State <> 8 OR DI2.State <> 8 OR DI3.State <> 8 OR DI4.State <> 8 OR AO1.State <> 8 OR AO2.State <> 8 OR DO1.State <> 8 OR DO2.State <> 8 OR DO3.State <> 8;

END_PROGRAM

// ---- POUs/0. Input/P0_02_AnalogInput.TcPOU
PROGRAM P0_02_AnalogInput
VAR PERSISTENT
	fbMixer_ActualSpeed			:FB_AnalogInput;
	fbMixer_ActualCurrent		:FB_AnalogInput;
	fbSieve_ActualSpeed			:FB_AnalogInput;
	fbChopper_ActualCurrent		:FB_AnalogInput;
	fbSP_ActualPressure			:FB_AnalogInput;
	fbSP_ActualSpeed			:FB_AnalogInput;
	fbSP_WaterTemperature		:FB_TemperatureInput;
	fbSP_LiquidTemperature		:FB_TemperatureInput;
END_VAR

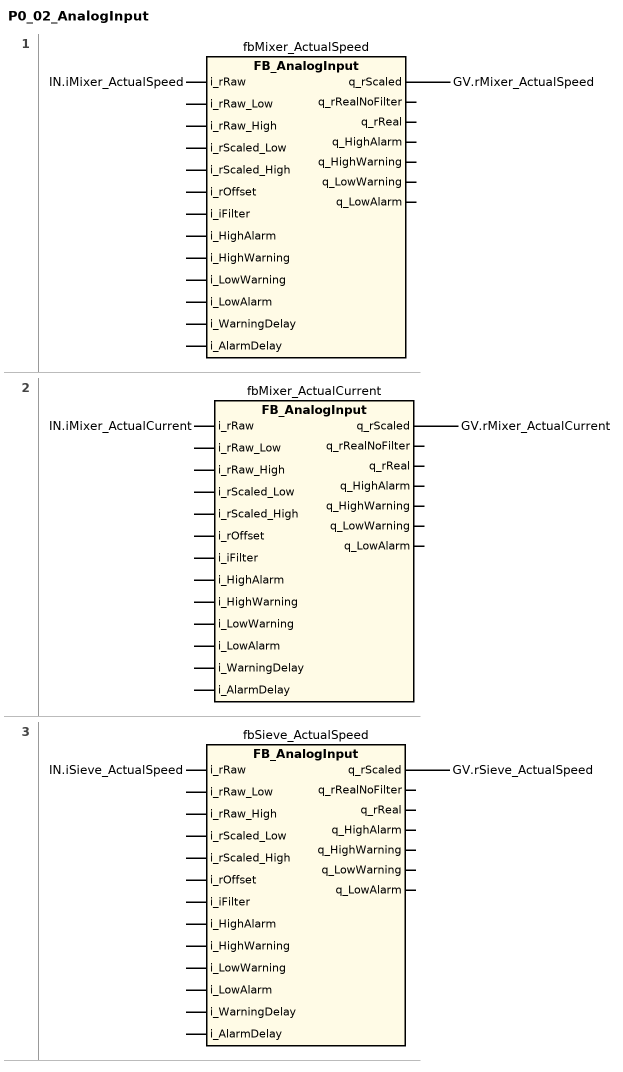
// NETWORK 1
fbMixer_ActualSpeed(i_rRaw := IN.iMixer_ActualSpeed); // FB_AnalogInput
GV.rMixer_ActualSpeed := fbMixer_ActualSpeed.q_rScaled;

// NETWORK 2
fbMixer_ActualCurrent(i_rRaw := IN.iMixer_ActualCurrent); // FB_AnalogInput
GV.rMixer_ActualCurrent := fbMixer_ActualCurrent.q_rScaled;

// NETWORK 3
fbSieve_ActualSpeed(i_rRaw := IN.iSieve_ActualSpeed); // FB_AnalogInput
GV.rSieve_ActualSpeed := fbSieve_ActualSpeed.q_rScaled;

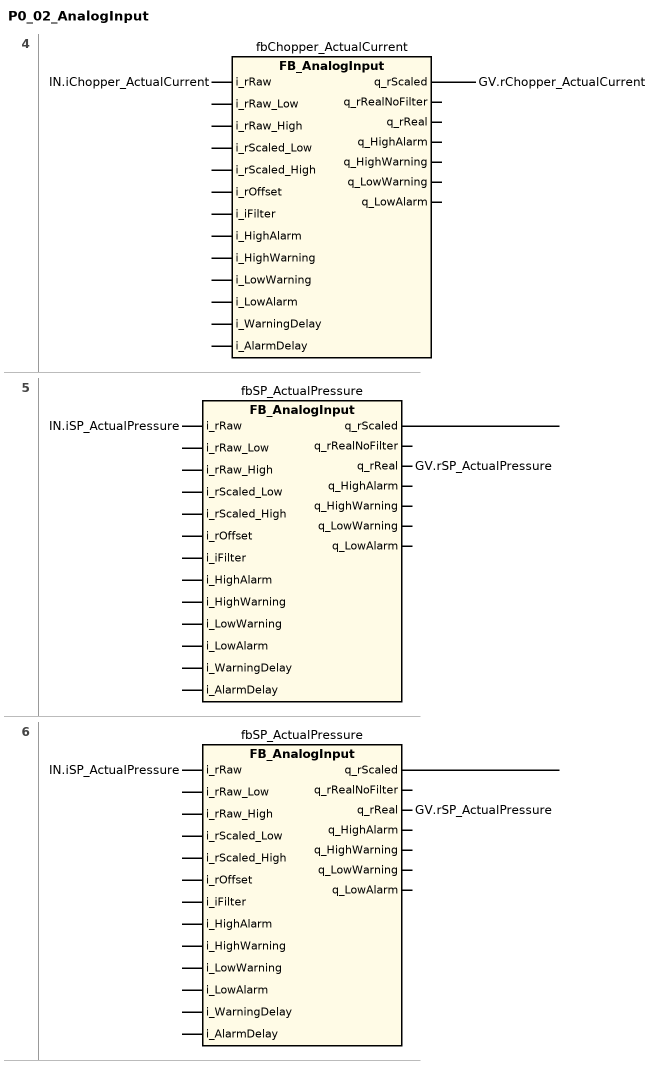
// NETWORK 4
fbChopper_ActualCurrent(i_rRaw := IN.iChopper_ActualCurrent); // FB_AnalogInput
GV.rChopper_ActualCurrent := fbChopper_ActualCurrent.q_rScaled;

// NETWORK 5
fbSP_ActualPressure(i_rRaw := IN.iSP_ActualPressure, q_rReal => GV.rSP_ActualPressure); // FB_AnalogInput

// NETWORK 6
fbSP_ActualPressure(i_rRaw := IN.iSP_ActualPressure, q_rReal => GV.rSP_ActualPressure); // FB_AnalogInput

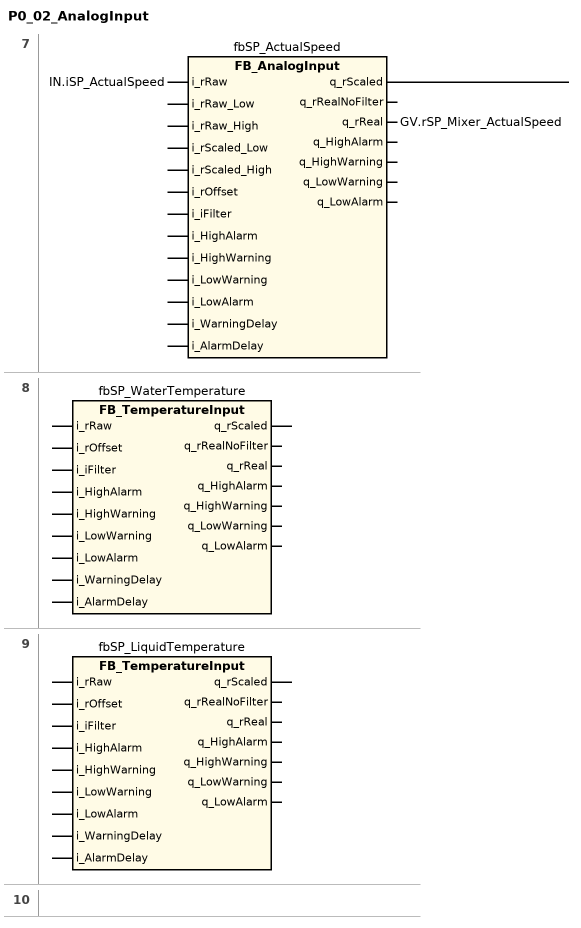
// NETWORK 7
fbSP_ActualSpeed(i_rRaw := IN.iSP_ActualSpeed, q_rReal => GV.rSP_Mixer_ActualSpeed); // FB_AnalogInput

// NETWORK 8
fbSP_WaterTemperature(); // FB_TemperatureInput

// NETWORK 9
fbSP_LiquidTemperature(); // FB_TemperatureInput

// NETWORK 10

END_PROGRAM

// ---- FBs/Devices/FB_AnalogInput.TcPOU
FUNCTION_BLOCK FB_AnalogInput
VAR_INPUT
	i_rRaw		 			:REAL;
	i_rRaw_Low				:REAL := 0;
	i_rRaw_High 			:REAL := 32767;
	i_rScaled_Low			:REAL := 0;
	i_rScaled_High			:REAL := 32767;
	i_rOffset 				:REAL;
	i_iFilter				:REAL  := 0.1;		//0-5s
	i_HighAlarm				:REAL;
	i_HighWarning			:REAL;
	i_LowWarning			:REAL;
	i_LowAlarm				:REAL;
	i_WarningDelay			:INT;
	i_AlarmDelay			:INT;
END_VAR
VAR_OUTPUT
	q_rScaled 				:REAL;
	q_rRealNoFilter			:REAL;
	q_rReal 				:REAL;
	q_HighAlarm				:BOOL;
	q_HighWarning			:BOOL;
	q_LowWarning			:BOOL;
	q_LowAlarm				:BOOL;
END_VAR
VAR
	K						:REAL;
	rRawInput				:REAL;
	tonHighAlarm			:TON;
	tonHighWarning			:TON;
	tonLowWarning			:TON;
	tonLowAlarm				:TON;
	arrSignals				:ARRAY[0..499] OF REAL;

	iLength					:INT;
	i						:INT;
	j						:INT;
	p						:INT;
	Sum						:REAL;
	
END_VAR

//Validation rules (protect divide by zero)
IF i_rRaw_High - i_rRaw_Low = 0 THEN
	i_rRaw_High := i_rRaw_Low + 1;
END_IF

//Scaling
K 				:= ((i_rScaled_High - i_rScaled_Low) /(i_rRaw_High - i_rRaw_Low));
rRawInput 		:= i_rRaw - i_rRaw_Low ;
q_rScaled 		:= (K * rRawInput) +  i_rScaled_Low;
q_rRealNoFilter	:= q_rScaled + i_rOffset;

//Filter
A_Filter();

//Warnings and alarms
tonHighAlarm(IN:=q_rReal>i_HighAlarm, PT:=INT_TO_TIME(i_AlarmDelay*1000));
tonHighWarning(IN:=q_rReal>i_HighWarning, PT:=INT_TO_TIME(i_WarningDelay*1000));
tonLowWarning(IN:=q_rReal<i_LowWarning, PT:=INT_TO_TIME(i_WarningDelay*1000));
tonLowAlarm(IN:=q_rReal<i_LowAlarm, PT:=INT_TO_TIME(i_AlarmDelay*1000));

q_HighAlarm := tonHighAlarm.Q;
q_HighWarning := tonHighWarning.Q;
q_LowWarning := tonLowWarning.Q;
q_LowAlarm := tonLowAlarm.Q;

//Warning and alarms validation rules
i_LowAlarm := LIMIT(i_rScaled_Low, i_LowAlarm, i_LowWarning);
i_HighAlarm := LIMIT(i_HighWarning, i_HighAlarm, i_rScaled_High);
i_LowWarning := LIMIT(i_LowAlarm, i_LowWarning, i_HighWarning);
i_HighWarning := LIMIT(i_LowWarning, i_HighWarning, i_HighAlarm);

ACTION A_Filter:
i_iFilter := LIMIT(0.1, i_iFilter, 5);
iLength := TO_INT(i_iFilter*100);

FOR p:=0 TO iLength-2 DO
	arrSignals[p]:=arrSignals[p+1];
END_FOR
arrSignals[iLength-1]:=q_rRealNoFilter;
Sum:=0;
FOR j:=0 TO iLength-1 DO
	Sum := Sum + arrSignals[j];
END_FOR
IF Sum <> 0 THEN
	q_rReal:=Sum/iLength;
ELSE
	q_rReal:=0;
END_IF
END_ACTION

//Created by MASAC Jan,2025

// Filter for analog signal (in seconds). Min filter time: 0s, Max filter time 5s
// Calculate average value of samples taken in last x seconds (if scan cycle remains 10ms)

METHOD M_Filter
VAR
	iLength				:INT;
	i					:INT;
	j					:INT;
	k					:INT;
	Sum					:REAL;
END_VAR
i_iFilter := LIMIT(0.1, i_iFilter, 5);
iLength := TO_INT(i_iFilter*100);

FOR k:=0 TO iLength-2 DO
	arrSignals[k]:=arrSignals[k+1];
END_FOR
arrSignals[iLength-1]:=q_rRealNoFilter;
Sum:=0;
FOR j:=0 TO iLength-1 DO
	Sum := Sum + arrSignals[j];
END_FOR
IF Sum <> 0 THEN
	q_rReal:=Sum/iLength;
END_IF
END_METHOD

END_FUNCTION_BLOCK

// ---- FBs/Devices/FB_TemperatureInput.TcPOU
FUNCTION_BLOCK FB_TemperatureInput
VAR_INPUT
	i_rRaw		 			:REAL;
	i_rOffset 				:REAL;
	i_iFilter				:REAL  := 0.1;		//0-5s
	i_HighAlarm				:REAL;
	i_HighWarning			:REAL;
	i_LowWarning			:REAL;
	i_LowAlarm				:REAL;
	i_WarningDelay			:INT;
	i_AlarmDelay			:INT;
END_VAR
VAR_OUTPUT
	q_rScaled 				:REAL;
	q_rRealNoFilter			:REAL;
	q_rReal 				:REAL;
	q_HighAlarm				:BOOL;
	q_HighWarning			:BOOL;
	q_LowWarning			:BOOL;
	q_LowAlarm				:BOOL;
END_VAR
VAR
	K						:INT :=10;
	tonHighAlarm			:TON;
	tonHighWarning			:TON;
	tonLowWarning			:TON;
	tonLowAlarm				:TON;
	arrSignals				:ARRAY[0..499] OF REAL;

END_VAR

//Scaling
q_rScaled 		:= i_rRaw/K;
q_rRealNoFilter	:= q_rScaled + i_rOffset;

//Filter
M_Filter();

//Warnings and alarms
tonHighAlarm(IN:=q_rReal>i_HighAlarm, PT:=INT_TO_TIME(i_AlarmDelay*1000));
tonHighWarning(IN:=q_rReal>i_HighWarning, PT:=INT_TO_TIME(i_WarningDelay*1000));
tonLowWarning(IN:=q_rReal<i_LowWarning, PT:=INT_TO_TIME(i_WarningDelay*1000));
tonLowAlarm(IN:=q_rReal<i_LowAlarm, PT:=INT_TO_TIME(i_AlarmDelay*1000));

q_HighAlarm := tonHighAlarm.Q;
q_HighWarning := tonHighWarning.Q;
q_LowWarning := tonLowWarning.Q;
q_LowAlarm := tonLowAlarm.Q;

// Filter for analog signal (in seconds). Min filter time: 0s, Max filter time 5s
// Calculate average value of samples taken in last x seconds (if scan cycle remains 10ms)

METHOD M_Filter
VAR
	iLength				:INT;
	i					:INT;
	j					:INT;
	k					:INT;
	Sum					:REAL;
END_VAR
i_iFilter := LIMIT(0.1, i_iFilter, 5);
iLength := TO_INT(i_iFilter*100);

FOR k:=0 TO iLength-2 DO
	arrSignals[k]:=arrSignals[k+1];
END_FOR
arrSignals[iLength-1]:=q_rRealNoFilter;
Sum:=0;
FOR j:=0 TO iLength-1 DO
	Sum := Sum + arrSignals[j];
END_FOR
IF Sum <> 0 THEN
	q_rReal:=Sum/iLength;
END_IF
END_METHOD

END_FUNCTION_BLOCK

// ---- POUs/1. Main Control/P1_00_MAIN.TcPOU
PROGRAM P1_00_MAIN
VAR
END_VAR

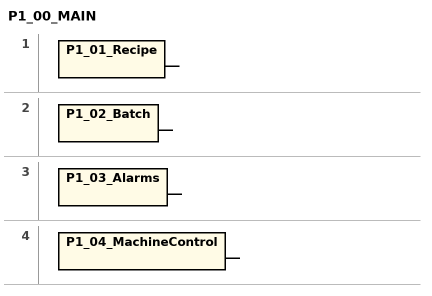
// NETWORK 1
P1_01_Recipe();

// NETWORK 2
P1_02_Batch();

// NETWORK 3
P1_03_Alarms();

// NETWORK 4
P1_04_MachineControl();

END_PROGRAM

// ---- POUs/1. Main Control/P1_01_Recipe.TcPOU
PROGRAM P1_01_Recipe
VAR
	i						:INT;
END_VAR

Recipes.Production.stPhase[1].bEnable:=TRUE;
Recipes.Production_Phase_HMI.bEnable:=TRUE;

Recipes.Cleaning.stPhase[1].bEnable:=TRUE;
Recipes.Cleaning_Phase_HMI.bEnable:=TRUE;

Recipes.Production.iActivePhase:=0;
Recipes.Cleaning.iActivePhase:=0;

FOR i := 1 TO 20 DO
	IF Recipes.Production.stPhase[i].bEnable THEN
		Recipes.Production.iActivePhase := i;
	END_IF
	
	IF NOT Recipes.Production.stPhase[i].bEnable THEN
		Recipes.Production.stPhase[i] := Recipes.Production_Empty.stPhase[0];
	END_IF
	
	IF Recipes.Cleaning.stPhase[i].bEnable THEN
		Recipes.Cleaning.iActivePhase := i;
	END_IF
	
	IF NOT Recipes.Cleaning.stPhase[i].bEnable THEN
		Recipes.Cleaning.stPhase[i] := Recipes.Cleaning_Empty.stPhase[0];
	END_IF
END_FOR

END_PROGRAM

// ---- POUs/1. Main Control/P1_02_Batch.TcPOU
PROGRAM P1_02_Batch
VAR
		fbBatch					:FB_Batch;
		fbBatchLog				:FB_BatchLog;
END_VAR
VAR PERSISTENT
	tonBatchTime				:FB_TONP;
END_VAR
VAR // added by the converter: edge detectors and wires of the graphical bodies
    _rt1, _rt2, _rt3, _rt4, _rt5, _rt6, _rt7, _rt8, _rt9, _rt10 : R_TRIG;
    _w1, _w2 : BOOL;
END_VAR

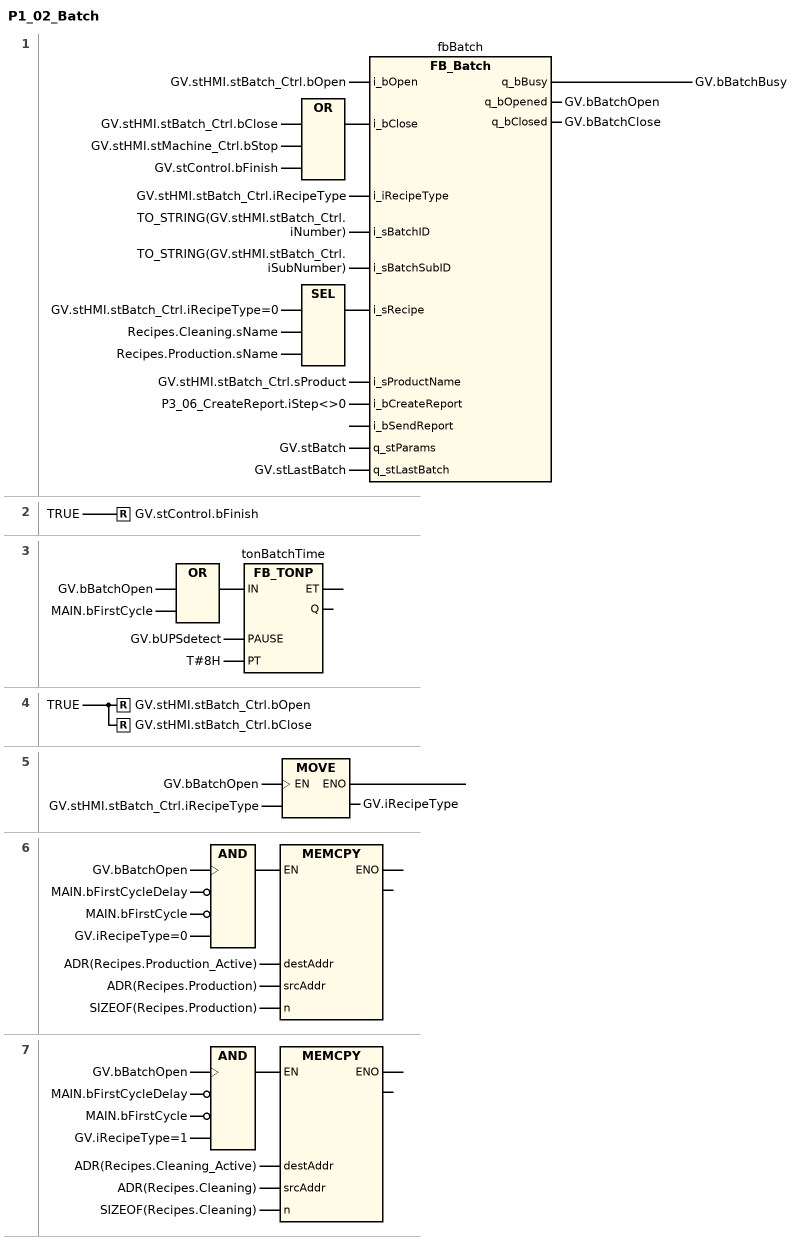
// NETWORK 1
fbBatch(
    i_bOpen := GV.stHMI.stBatch_Ctrl.bOpen,
    i_bClose := GV.stHMI.stBatch_Ctrl.bClose OR GV.stHMI.stMachine_Ctrl.bStop OR GV.stControl.bFinish,
    i_iRecipeType := GV.stHMI.stBatch_Ctrl.iRecipeType,
    i_sBatchID := TO_STRING(GV.stHMI.stBatch_Ctrl.iNumber),
    i_sBatchSubID := TO_STRING(GV.stHMI.stBatch_Ctrl.iSubNumber),
    i_sRecipe := SEL(GV.stHMI.stBatch_Ctrl.iRecipeType=0, Recipes.Cleaning.sName, Recipes.Production.sName),
    i_sProductName := GV.stHMI.stBatch_Ctrl.sProduct,
    i_bCreateReport := P3_06_CreateReport.iStep<>0,
    q_stParams := GV.stBatch,
    q_stLastBatch := GV.stLastBatch,
    q_bOpened => GV.bBatchOpen,
    q_bClosed => GV.bBatchClose); // FB_Batch
GV.bBatchBusy := fbBatch.q_bBusy;

// NETWORK 2
GV.stControl.bFinish R= TRUE;

// NETWORK 3
tonBatchTime(IN := GV.bBatchOpen OR MAIN.bFirstCycle, PAUSE := GV.bUPSdetect, PT := T#8H); // FB_TONP

// NETWORK 4
GV.stHMI.stBatch_Ctrl.bOpen R= TRUE;
GV.stHMI.stBatch_Ctrl.bClose R= TRUE;

// NETWORK 5
_rt1(CLK := GV.bBatchOpen);
IF _rt1.Q THEN GV.iRecipeType := GV.stHMI.stBatch_Ctrl.iRecipeType; END_IF

// NETWORK 6
_rt2(CLK := GV.bBatchOpen);
IF _rt2.Q AND NOT MAIN.bFirstCycleDelay AND NOT MAIN.bFirstCycle AND (GV.iRecipeType=0) THEN
    MEMCPY(destAddr := ADR(Recipes.Production_Active), srcAddr := ADR(Recipes.Production), n := SIZEOF(Recipes.Production));
END_IF

// NETWORK 7
_rt3(CLK := GV.bBatchOpen);
IF _rt3.Q AND NOT MAIN.bFirstCycleDelay AND NOT MAIN.bFirstCycle AND (GV.iRecipeType=1) THEN
    MEMCPY(destAddr := ADR(Recipes.Cleaning_Active), srcAddr := ADR(Recipes.Cleaning), n := SIZEOF(Recipes.Cleaning));
END_IF

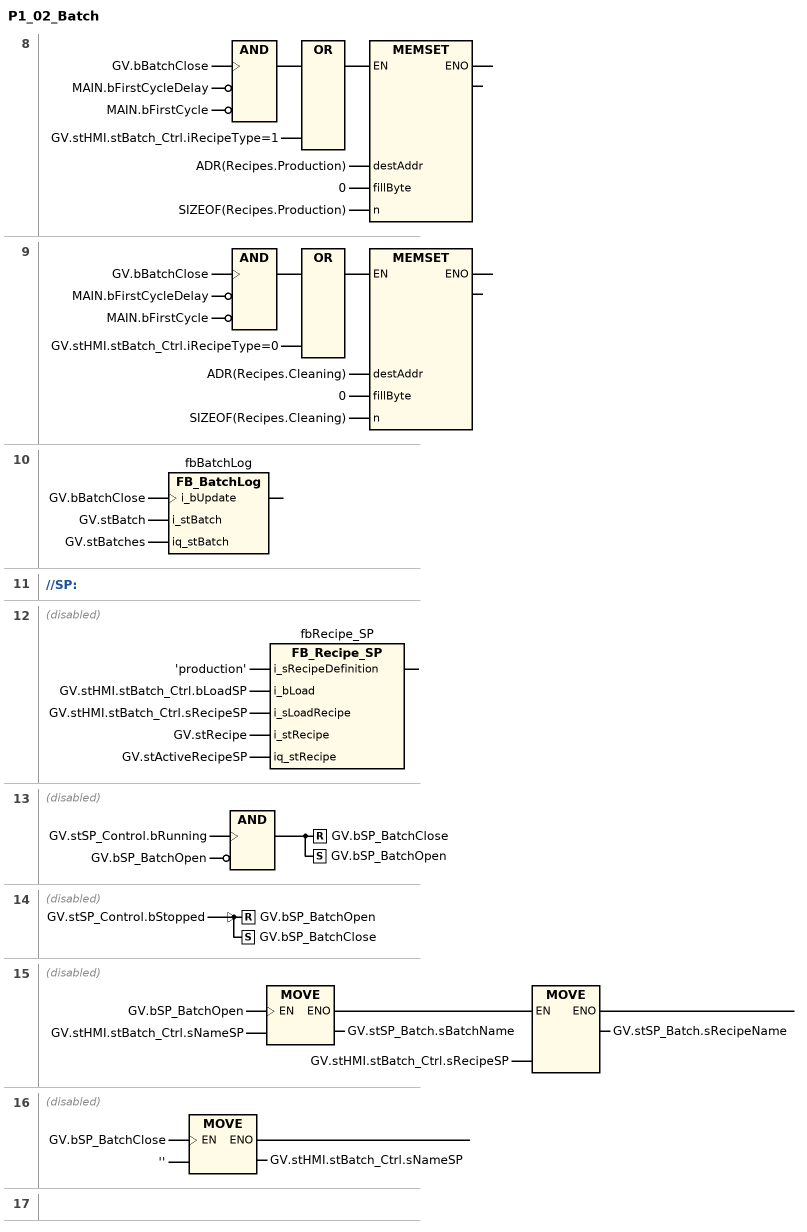
// NETWORK 8
_rt4(CLK := GV.bBatchClose);
IF _rt4.Q AND NOT MAIN.bFirstCycleDelay AND NOT MAIN.bFirstCycle OR (GV.stHMI.stBatch_Ctrl.iRecipeType=1) THEN
    MEMSET(destAddr := ADR(Recipes.Production), fillByte := 0, n := SIZEOF(Recipes.Production));
END_IF

// NETWORK 9
_rt5(CLK := GV.bBatchClose);
IF _rt5.Q AND NOT MAIN.bFirstCycleDelay AND NOT MAIN.bFirstCycle OR (GV.stHMI.stBatch_Ctrl.iRecipeType=0) THEN
    MEMSET(destAddr := ADR(Recipes.Cleaning), fillByte := 0, n := SIZEOF(Recipes.Cleaning));
END_IF

// NETWORK 10
_rt6(CLK := GV.bBatchClose);
fbBatchLog(i_bUpdate := _rt6.Q, i_stBatch := GV.stBatch, iq_stBatch := GV.stBatches); // FB_BatchLog

// NETWORK 11
// label: //SP

// NETWORK 12 (disabled)
// fbRecipe_SP(
//     i_sRecipeDefinition := 'production',
//     i_bLoad := GV.stHMI.stBatch_Ctrl.bLoadSP,
//     i_sLoadRecipe := GV.stHMI.stBatch_Ctrl.sRecipeSP,
//     i_stRecipe := GV.stRecipe,
//     iq_stRecipe := GV.stActiveRecipeSP); // FB_Recipe_SP

// NETWORK 13 (disabled)
// _rt7(CLK := GV.stSP_Control.bRunning);
// _w1 := _rt7.Q AND NOT GV.bSP_BatchOpen;
// GV.bSP_BatchClose R= _w1;
// GV.bSP_BatchOpen S= _w1;

// NETWORK 14 (disabled)
// _rt8(CLK := GV.stSP_Control.bStopped);
// GV.bSP_BatchOpen R= _rt8.Q;
// GV.bSP_BatchClose S= _rt8.Q;

// NETWORK 15 (disabled)
// _rt9(CLK := GV.bSP_BatchOpen);
// _w2 := _rt9.Q;
// IF _w2 THEN GV.stSP_Batch.sBatchName := GV.stHMI.stBatch_Ctrl.sNameSP; END_IF
// IF _w2 THEN GV.stSP_Batch.sRecipeName := GV.stHMI.stBatch_Ctrl.sRecipeSP; END_IF

// NETWORK 16 (disabled)
// _rt10(CLK := GV.bSP_BatchClose);
// IF _rt10.Q THEN GV.stHMI.stBatch_Ctrl.sNameSP := ''; END_IF

// NETWORK 17

END_PROGRAM

// ---- FBs/FB_Batch.TcPOU
FUNCTION_BLOCK FB_Batch
VAR_INPUT
	i_bOpen						:BOOL; 
	i_bClose					:BOOL; 
	i_iRecipeType				:INT;
	i_sBatchID					:STRING; 
	i_sBatchSubID				:STRING;
	i_sRecipe					:STRING;
	i_sProductName				:STRING;
	i_bCreateReport				:BOOL;
	i_bSendReport				:BOOL;
END_VAR
VAR_IN_OUT
	q_stParams					:ST_Batch;
	q_stLastBatch				:ST_Batch;
END_VAR
VAR_OUTPUT
	q_bBusy						:BOOL;	
	q_bOpened					:BOOL:=FALSE; 
	q_bClosed					:BOOL:=FALSE; 		
END_VAR

VAR
	tDelayCreateReport			:TON;
	tDelaySendReport			:TON;
	tDelayClose					:TON;
END_VAR	

VAR PERSISTENT
	iStep						:INT;
	sUserOpened					:STRING;
END_VAR

tDelayCreateReport(IN:=(iStep=200),PT:=T#3S);
tDelaySendReport(IN:=(iStep=300),PT:=T#3S);
tDelayClose(IN:=(iStep=110),PT:=T#500MS);

CASE iStep OF

	0: 
		MEMSET(ADR(q_stParams),0,SIZEOF(q_stParams));
		IF i_bOpen THEN
			iStep:=50;
		END_IF
		
	50:
		q_stParams.sRecipeType:=SEL(i_iRecipeType=0,'Cleaning','Production');
		IF i_sBatchSubID <> '0' THEN
			q_stParams.sBatchNumber:=CONCAT(i_sBatchID,'-');
			q_stParams.sBatchNumber:=CONCAT(q_stParams.sBatchNumber,i_sBatchSubID);
		ELSE
			q_stParams.sBatchNumber:=i_sBatchID;
		END_IF
		q_stParams.sRecipeName:=i_sRecipe;
		q_stParams.sProductName:=i_sProductName;
		q_stParams.sUser:=GV.sUserLogged;
		q_stParams.sStarted:=GV.stTime.sDateTime;
		sUserOpened:=GV.sUserLogged;
		iStep:=100;
			
	100:
		q_stParams.sUser:=sUserOpened;
		IF i_bClose THEN
			iStep:=110;
		END_IF
		
	110:
		IF tDelayClose.Q THEN
			q_stParams.sFinished:=GV.stTime.sDateTime;
			q_stLastBatch:=q_stParams;
			iStep:=200;
		END_IF
	200:
		IF tDelayCreateReport.Q AND NOT i_bCreateReport THEN
			iStep:=300;
		END_IF
	300:
		IF tDelaySendReport.Q AND NOT i_bSendReport THEN
			iStep:=1000;
		END_IF
		
	1000:
		iStep:=0;	
END_CASE

q_bBusy:=iStep<>0;
q_bOpened:=iStep=100;
q_bClosed:=iStep>110;

END_FUNCTION_BLOCK

// ---- FBs/FB_BatchLog.TcPOU
FUNCTION_BLOCK FB_BatchLog
VAR_INPUT
	i_bUpdate			:BOOL;
	i_stBatch			:ST_Batch;
END_VAR
VAR_IN_OUT
	iq_stBatch			:ARRAY[0..9] OF ST_Batch;
END_VAR
VAR
	i				:USINT;
	j				:USINT;
	bInsert			:BOOL;
END_VAR

IF i_bUpdate THEN
	bInsert:=FALSE;
	FOR i:=0 TO 9 DO
		IF iq_stBatch[i].sBatchNumber = '' THEN
			iq_stBatch[i]:=i_stBatch;
			bInsert:=TRUE;
			EXIT;
		END_IF
	END_FOR
	
	IF NOT bInsert THEN
		FOR j:=1 TO 9 DO
			iq_stBatch[j-1]:=iq_stBatch[j];
		END_FOR
		iq_stBatch[9]:=i_stBatch;
	END_IF
END_IF

END_FUNCTION_BLOCK

// ---- POUs/3. Report/P3_06_CreateReport.TcPOU
PROGRAM P3_06_CreateReport
VAR
	iStep					:INT;
	iError					:INT;
	tonResetError			:TON;
	trigStart				:R_TRIG;
	tonDelayStart			:TON;
	
	
	
	fbReport				:FB_PythonScript;
	fbSettingDelete			:FB_FileDelete;
	fbRecipeDelete			:FB_FileDelete;
	fbDeleteOldestBatch		:FB_DeleteOldestFile;
	fbSaveAsAlarm			:FB_FileSaveAs;
END_VAR


VAR PERSISTENT
	iReportsCreated			:INT;
END_VAR

ACT_CMDs();
tonResetError(IN:=(iError<>0),PT:=T#3S);
IF tonResetError.Q THEN
	iError:=0;
END_IF

trigStart(CLK:=GV.bBatchClose);

tonDelayStart(IN:=(iStep=10),PT:=T#1S);
CASE iStep OF
	
	0:
		IF trigStart.Q THEN
			iError:=0;
			iStep:=10;
		END_IF
		
	10:
		IF tonDelayStart.Q THEN
			iStep:=100;
		END_IF
		
	100:
		GV.stReport.bExport_Alarms:=TRUE;
		iStep:=110;
	110:
		IF NOT GV.stReport.bExport_Alarms THEN
			iStep:=200;
		END_IF
		
	200:
		GV.stReport.bCreate_Report:=TRUE;
		IF fbReport.q_bBusy THEN
			iStep:=210;
		END_IF
	210:
		IF NOT fbReport.q_bBusy AND fbReport.q_bDone THEN
			iStep:=400;
		ELSIF fbReport.q_bError THEN
			iError:=iStep;
			iStep:=999;
		END_IF
		
	400:
		IF GV.stBatches[9].sBatchNumber <> GV.sEmptyString THEN
			GV.stReport.bDelete_Data:=TRUE;
		END_IF
		iStep:=410;
	410:
		IF NOT GV.stReport.bDelete_Data THEN
			iStep:=500;
		END_IF;
	500:
		GV.stReport.bDelete_OldestReport:=TRUE;
		IF fbDeleteOldestBatch.q_bBusy THEN
			iStep:=510;
		END_IF
	510:
		IF NOT fbDeleteOldestBatch.q_bBusy AND fbDeleteOldestBatch.q_bDone THEN
			iStep:=900;
		ELSIF fbDeleteOldestBatch.q_bError THEN
			iStep:=900;
			iError:=iStep;
		END_IF
		
	900:
		iReportsCreated:=iReportsCreated+1;
		GV.stReport.bSend_Report:=TRUE;
		iStep:=0;
	999:
		iStep:=0;
END_CASE

ACTION ACT_CMDs:
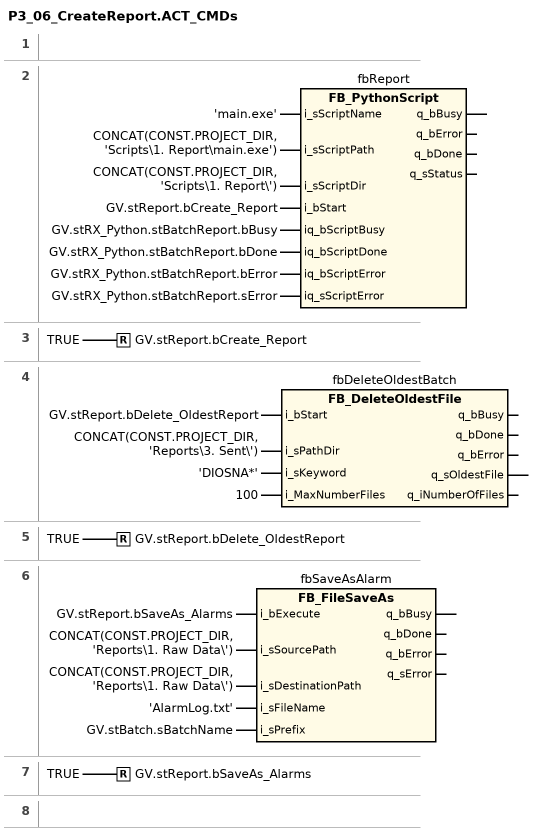
// NETWORK 1

// NETWORK 2
fbReport(
    i_sScriptName := 'main.exe',
    i_sScriptPath := CONCAT(CONST.PROJECT_DIR,'Scripts\1. Report\main.exe'),
    i_sScriptDir := CONCAT(CONST.PROJECT_DIR,'Scripts\1. Report\'),
    i_bStart := GV.stReport.bCreate_Report,
    iq_bScriptBusy := GV.stRX_Python.stBatchReport.bBusy,
    iq_bScriptDone := GV.stRX_Python.stBatchReport.bDone,
    iq_bScriptError := GV.stRX_Python.stBatchReport.bError,
    iq_sScriptError := GV.stRX_Python.stBatchReport.sError); // FB_PythonScript

// NETWORK 3
GV.stReport.bCreate_Report R= TRUE;

// NETWORK 4
fbDeleteOldestBatch(
    i_bStart := GV.stReport.bDelete_OldestReport,
    i_sPathDir := CONCAT(CONST.PROJECT_DIR,'Reports\3. Sent\'),
    i_sKeyword := 'DIOSNA*',
    i_MaxNumberFiles := 100); // FB_DeleteOldestFile

// NETWORK 5
GV.stReport.bDelete_OldestReport R= TRUE;

// NETWORK 6
fbSaveAsAlarm(
    i_bExecute := GV.stReport.bSaveAs_Alarms,
    i_sSourcePath := CONCAT(CONST.PROJECT_DIR,'Reports\1. Raw Data\'),
    i_sDestinationPath := CONCAT(CONST.PROJECT_DIR,'Reports\1. Raw Data\'),
    i_sFileName := 'AlarmLog.txt',
    i_sPrefix := GV.stBatch.sBatchName); // FB_FileSaveAs

// NETWORK 7
GV.stReport.bSaveAs_Alarms R= TRUE;

// NETWORK 8
END_ACTION

END_PROGRAM

// ---- FBs/FB_DeleteOldestFile.TcPOU
FUNCTION_BLOCK FB_DeleteOldestFile
VAR_INPUT
	i_bStart					:BOOL;
	i_sPathDir					:STRING[200];
	i_sKeyword					:STRING:='*';
	i_MaxNumberFiles			:UINT;
END_VAR
VAR_OUTPUT
	q_bBusy							:BOOL;
	q_bDone							:BOOL;
	q_bError						:BOOL;
	q_sOldestFile					:STRING;
	q_iNumberOfFiles				:UINT;
	
END_VAR
VAR
	fbFindFile				:FB_EnumFindFileEntry;
	eCmd					:E_EnumCmdType;
	bExecute				:BOOL;
	stFindFile				:ST_FindFileEntry;
	fbFileDelete			:FB_FileDelete;
	iStep					:INT:=0;
	sPath					:STRING[200];
	bDelete					:BOOL;
	sDeletePath				:STRING;
END_VAR

sPath:=CONCAT(i_sPathDir,i_sKeyword);
ACT_Files();
CASE iStep OF
	0:
		q_bBusy:=FALSE;
		IF i_bStart THEN
			q_iNumberOfFiles:=0;
			q_bDone:=FALSE;
			q_bError:=FALSE;
			q_bBusy:=TRUE;
			iStep:=10;
		END_IF
		
	10:
		eCmd := 0;
		bExecute:=TRUE;
		IF fbFindFile.bBusy THEN
			iStep:=20;
		END_IF
		
	20:
		IF NOT fbFindFile.bBusy THEN
			IF NOT fbFindFile.bError AND NOT fbFindFile.bEOE THEN
				q_sOldestFile:=stFindFile.sFileName;
				bExecute:=FALSE;
				iStep:=30;
			ELSIF NOT fbFindFile.bError AND fbFindFile.bEOE THEN
				bExecute:=FALSE;
				iStep:=100;
			ELSIF fbFindFile.bError THEN
				iStep:=999;
			END_IF
		END_IF
		
	30:
		q_iNumberOfFiles:=q_iNumberOfFiles+1;
		iStep:=40;
	
	40:
		eCmd := 1;
		bExecute:=TRUE;
		IF fbFindFile.bBusy THEN
			iStep:=50;
		END_IF
	
	50:
		IF NOT fbFindFile.bBusy THEN
			IF NOT fbFindFile.bError AND NOT fbFindFile.bEOE THEN
				bExecute:=FALSE;
				iStep:=30;
			ELSIF NOT fbFindFile.bError AND fbFindFile.bEOE THEN
				bExecute:=FALSE;
				iStep:=100;
			ELSIF fbFindFile.bError THEN
				iStep:=999;
			END_IF
		END_IF
		
	100:
		eCmd:=2;
		bExecute:=TRUE;
		IF NOT fbFindFile.bBusy THEN
			iStep:=150;
		END_IF
		
	150:
		IF q_iNumberOfFiles = i_MaxNumberFiles THEN
			iStep:=200;
		ELSE
			iStep:=300;
		END_IF
		
	200:
		sDeletePath:=CONCAT(i_sPathDir,q_sOldestFile);
		bDelete:=TRUE;
		iStep:=210;
	
	210:
		IF NOT fbFileDelete.bBusy THEN
			iStep:=300;
		END_IF
		
	300:
		q_bDone:=TRUE;
		iStep:=0;
		
	999:
		q_bError:=TRUE;
		iStep:=0;
		
		
END_CASE

ACTION ACT_Files:
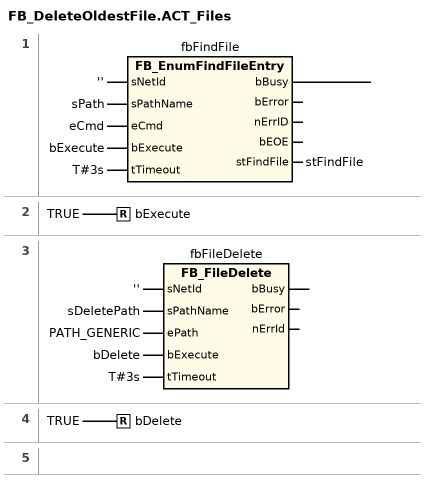
// NETWORK 1
fbFindFile(
    sNetId := '',
    sPathName := sPath,
    eCmd := eCmd,
    bExecute := bExecute,
    tTimeout := T#3s,
    stFindFile => stFindFile); // FB_EnumFindFileEntry

// NETWORK 2
bExecute R= TRUE;

// NETWORK 3
fbFileDelete(
    sNetId := '',
    sPathName := sDeletePath,
    ePath := PATH_GENERIC,
    bExecute := bDelete,
    tTimeout := T#3s); // FB_FileDelete

// NETWORK 4
bDelete R= TRUE;

// NETWORK 5
END_ACTION

END_FUNCTION_BLOCK

// ---- POUs/1. Main Control/P1_03_Alarms.TcPOU
PROGRAM P1_03_Alarms
VAR
	i					:USINT;
	bAlarmActive		:BOOL;
	bAlarmDisabled		:BOOL;
	TON_AlarmOK			:TON;

END_VAR
VAR PERSISTENT
	fbAlarm				:ARRAY [0..69] OF FB_AlarmDiagnostic;
END_VAR

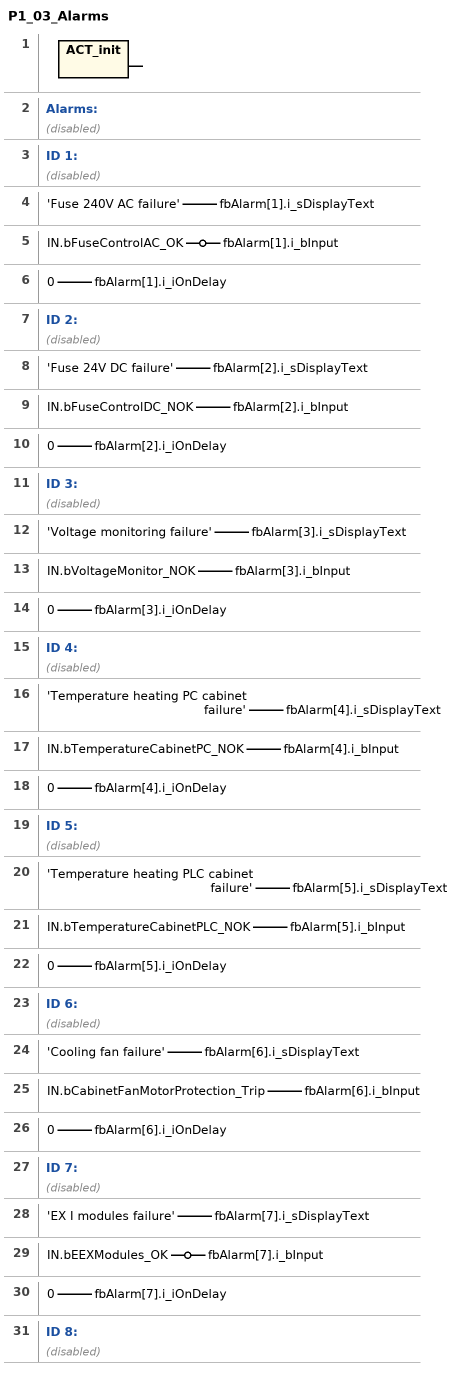
// NETWORK 1
ACT_init();

// NETWORK 2 (disabled)
// label: Alarms

// NETWORK 3 (disabled)
// label: ID 1

// NETWORK 4
fbAlarm[1].i_sDisplayText := 'Fuse 240V AC failure';

// NETWORK 5
fbAlarm[1].i_bInput := NOT IN.bFuseControlAC_OK;

// NETWORK 6
fbAlarm[1].i_iOnDelay := 0;

// NETWORK 7 (disabled)
// label: ID 2

// NETWORK 8
fbAlarm[2].i_sDisplayText := 'Fuse 24V DC failure';

// NETWORK 9
fbAlarm[2].i_bInput := IN.bFuseControlDC_NOK;

// NETWORK 10
fbAlarm[2].i_iOnDelay := 0;

// NETWORK 11 (disabled)
// label: ID 3

// NETWORK 12
fbAlarm[3].i_sDisplayText := 'Voltage monitoring failure';

// NETWORK 13
fbAlarm[3].i_bInput := IN.bVoltageMonitor_NOK;

// NETWORK 14
fbAlarm[3].i_iOnDelay := 0;

// NETWORK 15 (disabled)
// label: ID 4

// NETWORK 16
fbAlarm[4].i_sDisplayText := 'Temperature heating PC cabinet failure';

// NETWORK 17
fbAlarm[4].i_bInput := IN.bTemperatureCabinetPC_NOK;

// NETWORK 18
fbAlarm[4].i_iOnDelay := 0;

// NETWORK 19 (disabled)
// label: ID 5

// NETWORK 20
fbAlarm[5].i_sDisplayText := 'Temperature heating PLC cabinet failure';

// NETWORK 21
fbAlarm[5].i_bInput := IN.bTemperatureCabinetPLC_NOK;

// NETWORK 22
fbAlarm[5].i_iOnDelay := 0;

// NETWORK 23 (disabled)
// label: ID 6

// NETWORK 24
fbAlarm[6].i_sDisplayText := 'Cooling fan failure';

// NETWORK 25
fbAlarm[6].i_bInput := IN.bCabinetFanMotorProtection_Trip;

// NETWORK 26
fbAlarm[6].i_iOnDelay := 0;

// NETWORK 27 (disabled)
// label: ID 7

// NETWORK 28
fbAlarm[7].i_sDisplayText := 'EX I modules failure';

// NETWORK 29
fbAlarm[7].i_bInput := NOT IN.bEEXModules_OK;

// NETWORK 30
fbAlarm[7].i_iOnDelay := 0;

// NETWORK 31 (disabled)
// label: ID 8

